// TwinCAT 3 PLC project SPS_Demonstrator
// ProgramVersion: 3.1.4026.21
// libraries:
//   Tc2_Standard, * (Beckhoff Automation GmbH)
//   Tc2_System, * (Beckhoff Automation GmbH)
//   Tc3_EventLogger, * (Beckhoff Automation GmbH)
//   Tc3_Module, * (Beckhoff Automation GmbH)
// project tree:
//   GVLs/ GVL.TcGVL, GVL_HRL.TcGVL, GVL_HRL_Sim.TcGVL, GVL_MBS.TcGVL, GVL_Sim.TcGVL, GVL_SST.TcGVL, GVL_VSG.TcGVL, GVL_VSG_Sim.TcGVL, OPCUA.TcGVL
//   / PlcTask.TcTTO
//   POUs/AtomicSkillsSchablonen/ AutomaticColorDetection_nichtfertig.TcPOU, AxisControl_Encoder.TcPOU, AxisControl_MultipleInputSensors.TcPOU, CompressorControl.TcPOU, CuttingProcess.TcPOU, HardeningProcess.TcPOU, SecuringWorkpiece.TcPOU, StampingProcess.TcPOU
//   POUs/ControlOfOutputs/ HRL_ControlOfOutputs.TcPOU, MBS_ControlOfOutputs.TcPOU, SST_ControlOfOutputs.TcPOU, VSG_ControlOfOutputs.TcPOU
//   POUs/DiagnosisHandler/ HRL_DiagnosisHandler.TcPOU, VSG_DiagnosisHandler.TcPOU
//   POUs/ HRL_SkillSet.TcPOU, MBS_SkillSet.TcPOU, SST_SkillSet.TcPOU, VSG_SkillSet.TcPOU
//   POUs/InitStateDrive/ HRL_RGB_InitialStateDrive.TcPOU, MBS_DmPD_InitialStateDrive.TcPOU, MBS_MR01_InitialStateDrive.TcPOU, MBS_MR02_InitialStateDrive.TcPOU, MBS_VSG_InitialStateDrive.TcPOU, SST_PD_InitialStateDrive.TcPOU, VSG_InitialStateDrive.TcPOU
//   POUs/MethodenBeispiele/ FB_MyOpcUaMethod.TcPOU, JobMethode_Schablone.TcPOU
//   POUs/Moduls/HRL_Skills/ HRL_CB_AS_HorizontalMoveSensors.TcPOU, HRL_NMethod_Auslagern.TcPOU, HRL_RGB_AS_HorizontalMoveEncoders.TcPOU, HRL_RGB_AS_HorizontalMoveSensors.TcPOU, HRL_RGB_AS_VerticalMoveEncoders.TcPOU
//   POUs/Moduls/MBS_Skills/ MBS_CB_AS_HorizontalMove.TcPOU, MBS_DmPD_AS_HorizontalMove.TcPOU, MBS_DmPD_AS_RotationMove.TcPOU, MBS_MR01_AS_HardeningProcess.TcPOU, MBS_MR01_AS_HorizontalMoveSensors.TcPOU, MBS_MR01_AS_SecuringProcess.TcPOU, MBS_MR02_AS_CuttingProcess.TcPOU, MBS_VSG_AS_HorizontalMove.TcPOU, MBS_VSG_AS_SuctionProcess.TcPOU, MBS_VSG_AS_VerticalMove.TcPOU
//   POUs/Moduls/SST_Skills/ SST_CB_AS_HorizontalMove.TcPOU, SST_CS_AS_ColorDetection.TcPOU, SST_PD_AS_HorizontalMove.TcPOU
//   POUs/Moduls/VSG_Skills/ VSG_AS_CompressorControl.TcPOU, VSG_AS_HorizontalMoveEncoder.TcPOU, VSG_AS_RotationMoveEncoder.TcPOU, VSG_AS_VerticalMoveEncoder.TcPOU
//   POUs/OperatingModes/ HRL_OperatingModes.TcPOU, VSG_OperatingModes.TcPOU, MBS_OperatingModes.TcPOU, SST_OperatingModes.TcPOU, VSG_OperatingModes_alt.TcPOU
// real-time tasks:
//   TASK PlcTask: cycle T#10ms, priority 20, ADS port 350
// I/O:
//   DEVICE Gerät 1 (EtherCAT), AmsNetId 5.152.132.139.2.1
//     Klemme 1 (EK1200) [EK1200-5000 EtherCAT Netzteil (2A E-Bus)]
//       Klemme 2 (EL1512) [EL1512 2K. +/- Zaehler 24V, 1kHz]
//       Klemme 3 (EL1512) [EL1512 2K. +/- Zaehler 24V, 1kHz]
//       Klemme 4 (EL1512) [EL1512 2K. +/- Zaehler 24V, 1kHz]
//       Klemme 5 (EL1512) [EL1512 2K. +/- Zaehler 24V, 1kHz]
//       Klemme 6 (EL1512) [EL1512 2K. +/- Zaehler 24V, 1kHz]
//       Klemme 7 (EL1409) [EL1409 16K. Dig. Eingang 24V, 3ms]
//       Klemme 8 (EL1409) [EL1409 16K. Dig. Eingang 24V, 3ms]
//       Klemme 9 (EL2409) [EL2409 16K. Dig. Ausgang 24V, 0.5A]
//       Klemme 10 (EL2409) [EL2409 16K. Dig. Ausgang 24V, 0.5A]
//       Klemme 11 (EL2008) [EL2008 8K. Dig. Ausgang 24V, 0.5A]
//       Klemme 12 (EL3072) [EL3072 2K. Ana. Eingang  +/-10V, +/-20mA]
//       Klemme 13 (EL9011) [EL9011 Endklemme]
// variable links:
//   SPS_Demonstrator/SPS_Demonstrator Instance <-> Device 1 (EtherCAT)/Term 1 (EK1200)/Term 10 (EL2409)
//     PlcTask Outputs/GVL_MBS.MBS_Kompressor <-> Channel 2/Output
//     PlcTask Outputs/GVL_MBS.MBS_Leuchte_Ofen <-> Channel 1/Output
//     PlcTask Outputs/GVL_MBS.MBS_MV_Ofentuer <-> Channel 5/Output
//     PlcTask Outputs/GVL_MBS.MBS_MV_Schieber <-> Channel 6/Output
//     PlcTask Outputs/GVL_MBS.MBS_MV_Vakuum <-> Channel 3/Output
//     PlcTask Outputs/GVL_MBS.MBS_MV_senken <-> Channel 4/Output
//     PlcTask Outputs/GVL_SST.SST_Kompressor <-> Channel 16/Output
//     PlcTask Outputs/GVL_SST.SST_MOT_Foerderband <-> Channel 15/Output
//     PlcTask Outputs/GVL_VSG.VSG_Kompressor <-> Channel 13/Output
//     PlcTask Outputs/GVL_VSG.VSG_MOT_drehen_CCW <-> Channel 12/Output
//     PlcTask Outputs/GVL_VSG.VSG_MOT_drehen_CW <-> Channel 11/Output
//     PlcTask Outputs/GVL_VSG.VSG_MOT_horizontal_rueckwaerts <-> Channel 9/Output
//     PlcTask Outputs/GVL_VSG.VSG_MOT_horizontal_vorwaerts <-> Channel 10/Output
//     PlcTask Outputs/GVL_VSG.VSG_MOT_vertikal_hoch <-> Channel 7/Output
//     PlcTask Outputs/GVL_VSG.VSG_MOT_vertikal_runter <-> Channel 8/Output
//     PlcTask Outputs/GVL_VSG.VSG_MV_Vakuum <-> Channel 14/Output
//   SPS_Demonstrator/SPS_Demonstrator Instance <-> Device 1 (EtherCAT)/Term 1 (EK1200)/Term 11 (EL2008)
//     PlcTask Outputs/GVL_SST.SST_MV_blau <-> Channel 3/Output
//     PlcTask Outputs/GVL_SST.SST_MV_rot <-> Channel 2/Output
//     PlcTask Outputs/GVL_SST.SST_MV_weiss <-> Channel 1/Output
//   SPS_Demonstrator/SPS_Demonstrator Instance <-> Device 1 (EtherCAT)/Term 1 (EK1200)/Term 12 (EL3072)
//     PlcTask Inputs/GVL_SST.SST_Farbsensor <-> AI Standard Channel 1/Value
//   SPS_Demonstrator/SPS_Demonstrator Instance <-> Device 1 (EtherCAT)/Term 1 (EK1200)/Term 2 (EL1512)
//     PlcTask Inputs/GVL_HRL.HRL_Enc_horizontal_I1 <-> CNT Inputs Channel 1/Counter value
//     PlcTask Inputs/GVL_HRL.HRL_Enc_horizontal_I2 <-> CNT Inputs Channel 2/Counter value
//     PlcTask Outputs/GVL_HRL.HRL_K1_1_Zaehler_Zuruecksetzen <-> CNT Outputs Channel 1/Control/Set counter
//   SPS_Demonstrator/SPS_Demonstrator Instance <-> Device 1 (EtherCAT)/Term 1 (EK1200)/Term 3 (EL1512)
//     PlcTask Inputs/GVL_HRL.HRL_Enc_vertikal_I1 <-> CNT Inputs Channel 1/Counter value
//     PlcTask Inputs/GVL_HRL.HRL_Enc_vertikal_I2 <-> CNT Inputs Channel 2/Counter value
//     PlcTask Outputs/GVL_HRL.HRL_K1_2_Zaehler_Zuruecksetzen <-> CNT Outputs Channel 1/Control/Set counter
//   SPS_Demonstrator/SPS_Demonstrator Instance <-> Device 1 (EtherCAT)/Term 1 (EK1200)/Term 4 (EL1512)
//     PlcTask Inputs/GVL_VSG.VSG_Enc_vertikal_I1 <-> CNT Inputs Channel 1/Counter value
//     PlcTask Inputs/GVL_VSG.VSG_Enc_vertikal_I2 <-> CNT Inputs Channel 2/Counter value
//     PlcTask Outputs/GVL_VSG.VSG_K1_3_Zaehler_Zuruecksetzen <-> CNT Outputs Channel 1/Control/Set counter
//   SPS_Demonstrator/SPS_Demonstrator Instance <-> Device 1 (EtherCAT)/Term 1 (EK1200)/Term 5 (EL1512)
//     PlcTask Inputs/GVL_VSG.VSG_Enc_horizontal_I1 <-> CNT Inputs Channel 1/Counter value
//     PlcTask Inputs/GVL_VSG.VSG_Enc_horizontal_I2 <-> CNT Inputs Channel 2/Counter value
//     PlcTask Outputs/GVL_VSG.VSG_K1_4_Zaehler_Zuruecksetzen <-> CNT Outputs Channel 1/Set counter
//   SPS_Demonstrator/SPS_Demonstrator Instance <-> Device 1 (EtherCAT)/Term 1 (EK1200)/Term 6 (EL1512)
//     PlcTask Inputs/GVL_VSG.VSG_Enc_drehen_I1 <-> CNT Inputs Channel 1/Counter value
//     PlcTask Inputs/GVL_VSG.VSG_Enc_drehen_I2 <-> CNT Inputs Channel 2/Counter value
//     PlcTask Outputs/GVL_VSG.VSG_K1_5_Zaehler_Zuruecksetzen <-> CNT Outputs Channel 1/Control/Set counter
//   SPS_Demonstrator/SPS_Demonstrator Instance <-> Device 1 (EtherCAT)/Term 1 (EK1200)/Term 7 (EL1409)
//     PlcTask Inputs/GVL_HRL.HRL_LS_aussen <-> DIP Inputs/Input Channel 3
//     PlcTask Inputs/GVL_HRL.HRL_LS_innen <-> DIP Inputs/Input Channel 2
//     PlcTask Inputs/GVL_HRL.HRL_Ref_Taster_Ausleger_hinten <-> DIP Inputs/Input Channel 8
//     PlcTask Inputs/GVL_HRL.HRL_Ref_Taster_Ausleger_vorne <-> DIP Inputs/Input Channel 7
//     PlcTask Inputs/GVL_HRL.HRL_Ref_Taster_horizontal <-> DIP Inputs/Input Channel 1
//     PlcTask Inputs/GVL_HRL.HRL_Ref_Taster_vertikal <-> DIP Inputs/Input Channel 4
//     PlcTask Inputs/GVL_HRL.HRL_Spursensor_1_unten <-> DIP Inputs/Input Channel 5
//     PlcTask Inputs/GVL_HRL.HRL_Spursensor_2_oben <-> DIP Inputs/Input Channel 6
//     PlcTask Inputs/GVL_MBS.MBS_LS_Ende_Foerderband <-> DIP Inputs/Input Channel 11
//     PlcTask Inputs/GVL_MBS.MBS_Ref_Taster_DK_Pos_Foerderband <-> DIP Inputs/Input Channel 10
//     PlcTask Inputs/GVL_MBS.MBS_Ref_Taster_DK_Pos_Saege <-> DIP Inputs/Input Channel 12
//     PlcTask Inputs/GVL_MBS.MBS_Ref_Taster_DK_Pos_Sauger <-> DIP Inputs/Input Channel 9
//     PlcTask Inputs/GVL_MBS.MBS_Ref_Taster_Ofenschieber_aussen <-> DIP Inputs/Input Channel 15
//     PlcTask Inputs/GVL_MBS.MBS_Ref_Taster_Ofenschieber_innen <-> DIP Inputs/Input Channel 14
//     PlcTask Inputs/GVL_MBS.MBS_Ref_Taster_Sauger_Pos_DK <-> DIP Inputs/Input Channel 13
//     PlcTask Inputs/GVL_MBS.MBS_Ref_Taster_Sauger_Pos_Ofen <-> DIP Inputs/Input Channel 16
//   SPS_Demonstrator/SPS_Demonstrator Instance <-> Device 1 (EtherCAT)/Term 1 (EK1200)/Term 8 (EL1409)
//     PlcTask Inputs/GVL.diNotAus_Kanal_A <-> DIP Inputs/Input Channel 11
//     PlcTask Inputs/GVL.diNotAus_Kanal_B <-> DIP Inputs/Input Channel 12
//     PlcTask Inputs/GVL_MBS.MBS_LS_Ofen <-> DIP Inputs/Input Channel 1
//     PlcTask Inputs/GVL_SST.SST_Impulstaster <-> DIP Inputs/Input Channel 5
//     PlcTask Inputs/GVL_SST.SST_LS_Eingang <-> DIP Inputs/Input Channel 6
//     PlcTask Inputs/GVL_SST.SST_LS_blau <-> DIP Inputs/Input Channel 10
//     PlcTask Inputs/GVL_SST.SST_LS_nach_Farbsensor <-> DIP Inputs/Input Channel 7
//     PlcTask Inputs/GVL_SST.SST_LS_rot <-> DIP Inputs/Input Channel 9
//     PlcTask Inputs/GVL_SST.SST_LS_weiss <-> DIP Inputs/Input Channel 8
//     PlcTask Inputs/GVL_VSG.VSG_Ref_Schalter_drehen <-> DIP Inputs/Input Channel 4
//     PlcTask Inputs/GVL_VSG.VSG_Ref_Schalter_horizontal <-> DIP Inputs/Input Channel 3
//     PlcTask Inputs/GVL_VSG.VSG_Ref_Schalter_vertikal <-> DIP Inputs/Input Channel 2
//   SPS_Demonstrator/SPS_Demonstrator Instance <-> Device 1 (EtherCAT)/Term 1 (EK1200)/Term 9 (EL2409)
//     PlcTask Outputs/GVL_HRL.HRL_MOT_Ausleger_rueckwaerts <-> Channel 8/Output
//     PlcTask Outputs/GVL_HRL.HRL_MOT_Ausleger_vorwaerts <-> Channel 7/Output
//     PlcTask Outputs/GVL_HRL.HRL_MOT_Foerderband_rueckwaerts <-> Channel 2/Output
//     PlcTask Outputs/GVL_HRL.HRL_MOT_Foerderband_vorwaerts <-> Channel 1/Output
//     PlcTask Outputs/GVL_HRL.HRL_MOT_horizontal_zum_Foerderband <-> Channel 4/Output
//     PlcTask Outputs/GVL_HRL.HRL_MOT_horizontal_zum_Regal <-> Channel 3/Output
//     PlcTask Outputs/GVL_HRL.HRL_MOT_vertikal_hoch <-> Channel 6/Output
//     PlcTask Outputs/GVL_HRL.HRL_MOT_vertikal_runter <-> Channel 5/Output
//     PlcTask Outputs/GVL_MBS.MBS_MOT_DK_CCW <-> Channel 10/Output
//     PlcTask Outputs/GVL_MBS.MBS_MOT_DK_CW <-> Channel 9/Output
//     PlcTask Outputs/GVL_MBS.MBS_MOT_Foerderband_vorwaerts <-> Channel 11/Output
//     PlcTask Outputs/GVL_MBS.MBS_MOT_Ofenschieber_ausfahren <-> Channel 14/Output
//     PlcTask Outputs/GVL_MBS.MBS_MOT_Ofenschieber_einfahren <-> Channel 13/Output
//     PlcTask Outputs/GVL_MBS.MBS_MOT_Saege <-> Channel 12/Output
//     PlcTask Outputs/GVL_MBS.MBS_MOT_Sauger_zum_DK <-> Channel 16/Output
//     PlcTask Outputs/GVL_MBS.MBS_MOT_Sauger_zum_Ofen <-> Channel 15/Output

CONFIGURATION SPS_Demonstrator
    RESOURCE PLC ON TwinCAT3
        TASK PlcTask(INTERVAL := T#10ms, PRIORITY := 20);
        PROGRAM HRL_SkillSet WITH PlcTask : HRL_SkillSet;
        PROGRAM VSG_SkillSet WITH PlcTask : VSG_SkillSet;
    END_RESOURCE
END_CONFIGURATION

// ---- GVLs/GVL.TcGVL
{attribute 'qualified_only'}
VAR_GLOBAL
	// xDI%139.2_S1_2
	diNotAus_Kanal_A AT %I*: BOOL;
	// xDI%139.3_S1_2
	diNotAus_Kanal_B AT %I*: BOOL;
END_VAR

// ---- GVLs/GVL_HRL.TcGVL
{attribute 'qualified_only'}
VAR_GLOBAL
	// udiDI%41.0_A2_5
	{attribute 'OPC.UA.DA' := '1'} // für OPC UA freigeben
	HRL_Enc_horizontal_I1 AT %I*: UDINT;
	{attribute 'OPC.UA.DA' := '1'} // für OPC UA freigeben
	// udiDI%47.0_A2_5
	HRL_Enc_horizontal_I2 AT %I*: UDINT;
	{attribute 'OPC.UA.DA' := '1'} // für OPC UA freigeben
	// udiDI%53.0_A2_5
	HRL_Enc_vertikal_I1 AT %I*: UDINT;
	{attribute 'OPC.UA.DA' := '1'} // für OPC UA freigeben
	// udiDI%59.0_A2_5
	HRL_Enc_vertikal_I2 AT %I*: UDINT;
	{attribute 'OPC.UA.DA' := '1'} // für OPC UA freigeben
	// xDI%136.0_A2_2
	HRL_Ref_Taster_horizontal AT %I*: BOOL;
	{attribute 'OPC.UA.DA' := '1'} // für OPC UA freigeben
	// xDI%136.1_A2_1
	{attribute 'OPC.UA.DA' := '1'} // für OPC UA freigeben
	HRL_LS_innen AT %I*: BOOL;
	// xDI%136.2_A2_1
	{attribute 'OPC.UA.DA' := '1'} // für OPC UA freigeben
	HRL_LS_aussen AT %I*: BOOL;
	// xDI%136.3_A2_2
	{attribute 'OPC.UA.DA' := '1'} // für OPC UA freigeben
	HRL_Ref_Taster_vertikal AT %I*: BOOL;
	// xDI%136.4_A2_3
	{attribute 'OPC.UA.DA' := '1'} // für OPC UA freigeben
	HRL_Spursensor_1_unten AT %I*: BOOL;
	// xDI%136.5_A2_3
	{attribute 'OPC.UA.DA' := '1'} // für OPC UA freigeben
	HRL_Spursensor_2_oben AT %I*: BOOL;
	// xDI%136.6_A2_2
	{attribute 'OPC.UA.DA' := '1'} // für OPC UA freigeben
	HRL_Ref_Taster_Ausleger_vorne AT %I*: BOOL;
	// xDI%136.7_A2_2
	{attribute 'OPC.UA.DA' := '1'} // für OPC UA freigeben
	HRL_Ref_Taster_Ausleger_hinten AT %I*: BOOL;
	// xDO%111.0_A2_2	
	{attribute 'OPC.UA.DA' := '1'} // für OPC UA freigeben
	HRL_MOT_Foerderband_vorwaerts AT %Q*: BOOL;
	// xDO%111.1_A2_2
	{attribute 'OPC.UA.DA' := '1'} // für OPC UA freigeben
	HRL_MOT_Foerderband_rueckwaerts AT %Q*: BOOL;
	// xDO%111.2_A2_4
	{attribute 'OPC.UA.DA' := '1'} // für OPC UA freigeben
	HRL_MOT_horizontal_zum_Regal AT %Q*: BOOL;
	// xDO%111.3_A2_4
	{attribute 'OPC.UA.DA' := '1'} // für OPC UA freigeben
	HRL_MOT_horizontal_zum_Foerderband AT %Q*: BOOL;
	// xDO%111.4_A2_4
	{attribute 'OPC.UA.DA' := '1'} // für OPC UA freigeben
	HRL_MOT_vertikal_runter AT %Q*: BOOL;
	// xDO%111.5_A2_4
	{attribute 'OPC.UA.DA' := '1'} // für OPC UA freigeben
	HRL_MOT_vertikal_hoch AT %Q*: BOOL;
	// xDO%111.6_A2_4
	{attribute 'OPC.UA.DA' := '1'} // für OPC UA freigeben
	HRL_MOT_Ausleger_vorwaerts AT %Q*: BOOL;
	// xDO%111.7_A2_4
	{attribute 'OPC.UA.DA' := '1'} // für OPC UA freigeben
	HRL_MOT_Ausleger_rueckwaerts AT %Q*: BOOL;
	{attribute 'OPC.UA.DA' := '1'} // für OPC UA freigeben
	HRL_K1_1_Zaehler_Zuruecksetzen AT %Q*: BOOL;
	{attribute 'OPC.UA.DA' := '1'} // für OPC UA freigeben
	HRL_K1_2_Zaehler_Zuruecksetzen AT %Q*: BOOL;
END_VAR

// ---- GVLs/GVL_HRL_Sim.TcGVL
{attribute 'qualified_only'}
VAR_GLOBAL
	// Spiegel von GVL_HRL (Eingänge)
    HRL_Enc_horizontal_I1 : UDINT;
	// udiDI%47.0_A2_5
	HRL_Enc_horizontal_I2 : UDINT;
	// udiDI%53.0_A2_5
	HRL_Enc_vertikal_I1 : UDINT;
	// udiDI%59.0_A2_5
	HRL_Enc_vertikal_I2 : UDINT;
	// xDI%136.0_A2_2
	HRL_Ref_Taster_horizontal : BOOL;
	// xDI%136.1_A2_1
	HRL_LS_innen : BOOL;
	// xDI%136.2_A2_1
	HRL_LS_aussen : BOOL;
	// xDI%136.3_A2_2
	HRL_Ref_Taster_vertikal : BOOL;
	// xDI%136.4_A2_3
	HRL_Spursensor_1_unten : BOOL;
	// xDI%136.5_A2_3
	HRL_Spursensor_2_oben : BOOL;
	// xDI%136.6_A2_2
	HRL_Ref_Taster_Ausleger_vorne : BOOL;
	// xDI%136.7_A2_2
	HRL_Ref_Taster_Ausleger_hinten : BOOL;
	// xDO%111.0_A2_2	
	HRL_MOT_Foerderband_vorwaerts : BOOL;
	// xDO%111.1_A2_2
	HRL_MOT_Foerderband_rueckwaerts : BOOL;
	// xDO%111.2_A2_4
	HRL_MOT_horizontal_zum_Regal : BOOL;
	// xDO%111.3_A2_4
	HRL_MOT_horizontal_zum_Foerderband : BOOL;
	// xDO%111.4_A2_4
	HRL_MOT_vertikal_runter : BOOL;
	// xDO%111.5_A2_4
	HRL_MOT_vertikal_hoch : BOOL;
	// xDO%111.6_A2_4
	HRL_MOT_Ausleger_vorwaerts : BOOL;
	// xDO%111.7_A2_4
	HRL_MOT_Ausleger_rueckwaerts : BOOL;
	HRL_K1_1_Zaehler_Zuruecksetzen : BOOL;
	HRL_K1_2_Zaehler_Zuruecksetzen : BOOL;
END_VAR

// ---- GVLs/GVL_MBS.TcGVL
{attribute 'qualified_only'}
VAR_GLOBAL
	// xDI%137.0_A3_2
	MBS_Ref_Taster_DK_Pos_Sauger AT %I*: BOOL;
	// xDI%137.1_A3_2
	MBS_Ref_Taster_DK_Pos_Foerderband AT %I*: BOOL;
	// xDI%137.2_A3_1
	MBS_LS_Ende_Foerderband AT %I*: BOOL;
	// xDI%137.3_A3_2
	MBS_Ref_Taster_DK_Pos_Saege AT %I*: BOOL;
	// xDI%137.4_A3_2
	MBS_Ref_Taster_Sauger_Pos_DK AT %I*: BOOL;
	// xDI%137.5_A3_2
	MBS_Ref_Taster_Ofenschieber_innen AT %I*: BOOL;
	// xDI%137.6_A3_2
	MBS_Ref_Taster_Ofenschieber_aussen AT %I*: BOOL;
	// xDI%137.7_A3_2
	MBS_Ref_Taster_Sauger_Pos_Ofen AT %I*: BOOL;
	// xDI%138.0_A3_1
	MBS_LS_Ofen AT %I*: BOOL;
	// xDO%112.0_A3_4
	MBS_MOT_DK_CW AT %Q*: BOOL;
	// xDO%112.1_A3_4
	MBS_MOT_DK_CCW AT %Q*: BOOL;
	// xDO%112.2_A3_2
	MBS_MOT_Foerderband_vorwaerts AT %Q*: BOOL;
	// xDO%112.3_A3_6
	MBS_MOT_Saege AT %Q*: BOOL;
	// xDO%112.4_A3_3
	MBS_MOT_Ofenschieber_einfahren AT %Q*: BOOL;
	// xDO%112.5_A3_3
	MBS_MOT_Ofenschieber_ausfahren AT %Q*: BOOL;
	// xDO%112.6_A3_5
	MBS_MOT_Sauger_zum_Ofen AT %Q*: BOOL;
	// xDO%112.7_A3_5
	MBS_MOT_Sauger_zum_DK AT %Q*: BOOL;
	// xDO%113.0_A3_7
	MBS_Leuchte_Ofen AT %Q*: BOOL;
	// xDO%113.1_A3_8
	MBS_Kompressor AT %Q*: BOOL;
	// xDO%113.2_A3_5
	MBS_MV_Vakuum AT %Q*: BOOL;
	// xDO%113.3_A3_5
	MBS_MV_senken AT %Q*: BOOL;
	// xDO%113.4_A3_5
	MBS_MV_Ofentuer AT %Q*: BOOL;
	// xDO%113.5_A3_5
	MBS_MV_Schieber AT %Q*: BOOL;
END_VAR

// ---- GVLs/GVL_Sim.TcGVL
{attribute 'qualified_only'}
VAR_GLOBAL
	bSimMode : BOOL ;   // FALSE = reale Hardware, TRUE = Python-Simulation

    // Spiegel von GVL
    diNotAus_Kanal_A : BOOL ;
    diNotAus_Kanal_B : BOOL ;
    
END_VAR

// ---- GVLs/GVL_SST.TcGVL
{attribute 'qualified_only'}
VAR_GLOBAL
	// xDO%115.0_A5_5
	SST_MV_weiss AT %Q*: BOOL;
	// xDO%115.1_A5_5
	SST_MV_rot AT %Q*: BOOL;
	// xDO%115.2_A5_5
	SST_MV_blau AT %Q*: BOOL;
	// iAI%130.0_A5_4
	SST_Farbsensor AT %I*: INT;
	// xDI%138.4_A5_1
	SST_Impulstaster AT %I*: BOOL;
	// xDI%138.5_A5_1
	SST_LS_Eingang AT %I*: BOOL;
	// xDI%138.6_A5_1
	SST_LS_nach_Farbsensor AT %I*: BOOL;
	// xDI%138.7_A5_1
	SST_LS_weiss AT %I*: BOOL;
	// xDI%139.0_A5_1
	SST_LS_rot AT %I*: BOOL;
	// xDI%139.1_A5_1
	SST_LS_blau AT %I*: BOOL;
	// xDO%114.6_A5_2
	SST_MOT_Foerderband AT %Q*: BOOL;
	// xDO%114.7_A5_8
	SST_Kompressor AT %Q*: BOOL;
END_VAR

// ---- GVLs/GVL_VSG.TcGVL
{attribute 'qualified_only'}
VAR_GLOBAL
	// udiDI%65.0_A4_5
	{attribute 'OPC.UA.DA' := '1'} // für OPC UA freigeben
	VSG_Enc_vertikal_I1 AT %I*: UDINT;
	{attribute 'OPC.UA.DA' := '1'} // für OPC UA freigeben
	// udiDI%71.0_A4_5
	VSG_Enc_vertikal_I2 AT %I*: UDINT;
	{attribute 'OPC.UA.DA' := '1'} // für OPC UA freigeben
	// udiDI%77.0_A4_5
	VSG_Enc_horizontal_I1 AT %I*: UDINT;
	{attribute 'OPC.UA.DA' := '1'} // für OPC UA freigeben
	// udiDI%83.0_A4_5
	VSG_Enc_horizontal_I2 AT %I*: UDINT;
	{attribute 'OPC.UA.DA' := '1'} // für OPC UA freigeben
	// udiDI%89.0_A4_5
	VSG_Enc_drehen_I1 AT %I*: UDINT;
	{attribute 'OPC.UA.DA' := '1'} // für OPC UA freigeben
	// udiDI%95.0_A4_5
	VSG_Enc_drehen_I2 AT %I*: UDINT;
	{attribute 'OPC.UA.DA' := '1'} // für OPC UA freigeben
	// xDI%138.1_A4_2
	VSG_Ref_Schalter_vertikal AT %I*: BOOL;
	{attribute 'OPC.UA.DA' := '1'} // für OPC UA freigeben
	// xDI%138.2_A4_2
	VSG_Ref_Schalter_horizontal AT %I*: BOOL;
	{attribute 'OPC.UA.DA' := '1'} // für OPC UA freigeben
	// xDI%138.3_A4_2
	VSG_Ref_Schalter_drehen AT %I*: BOOL;
	{attribute 'OPC.UA.DA' := '1'} // für OPC UA freigeben
	// xDO%113.6_A4_4
	VSG_MOT_vertikal_hoch AT %Q*: BOOL;
	{attribute 'OPC.UA.DA' := '1'} // für OPC UA freigeben
	// xDO%113.7_A4_4
	VSG_MOT_vertikal_runter AT %Q*: BOOL;
	{attribute 'OPC.UA.DA' := '1'} // für OPC UA freigeben
	// xDO%114.0_A4_4
	VSG_MOT_horizontal_rueckwaerts AT %Q*: BOOL;
	{attribute 'OPC.UA.DA' := '1'} // für OPC UA freigeben
	// xDO%114.1_A4_4
	VSG_MOT_horizontal_vorwaerts AT %Q*: BOOL;
	{attribute 'OPC.UA.DA' := '1'} // für OPC UA freigeben
	// xDO%114.2_A4_4
	VSG_MOT_drehen_CW AT %Q*: BOOL;
	{attribute 'OPC.UA.DA' := '1'} // für OPC UA freigeben
	// xDO%114.3_A4_4
	VSG_MOT_drehen_CCW AT %Q*: BOOL;
	{attribute 'OPC.UA.DA' := '1'} // für OPC UA freigeben
	// xDO%114.4_A4_8
	VSG_Kompressor AT %Q*: BOOL;
	{attribute 'OPC.UA.DA' := '1'} // für OPC UA freigeben
	// xDO%114.5_A4_5
	{attribute 'OPC.UA.DA' := '1'} // für OPC UA freigeben
	VSG_MV_Vakuum AT %Q*: BOOL;
	{attribute 'OPC.UA.DA' := '1'} // für OPC UA freigeben
	VSG_K1_4_Zaehler_Zuruecksetzen AT %Q*: BOOL;
	{attribute 'OPC.UA.DA' := '1'} // für OPC UA freigeben
	VSG_K1_5_Zaehler_Zuruecksetzen AT %Q*: BOOL;
	{attribute 'OPC.UA.DA' := '1'} // für OPC UA freigeben
	VSG_K1_3_Zaehler_Zuruecksetzen AT %Q*: BOOL;
END_VAR

// ---- GVLs/GVL_VSG_Sim.TcGVL
{attribute 'qualified_only'}
VAR_GLOBAL
    // Simulierte VSG Eingänge
    VSG_Enc_vertikal_I1 : UDINT;
    VSG_Enc_vertikal_I2 : UDINT;

    VSG_Enc_horizontal_I1 : UDINT;
    VSG_Enc_horizontal_I2 : UDINT;

    VSG_Enc_drehen_I1 : UDINT;
    VSG_Enc_drehen_I2 : UDINT;

    VSG_Ref_Schalter_vertikal : BOOL;
    VSG_Ref_Schalter_horizontal : BOOL;
    VSG_Ref_Schalter_drehen : BOOL;

    // Simulierte VSG Ausgänge
    VSG_MOT_vertikal_hoch : BOOL;
    VSG_MOT_vertikal_runter : BOOL;

    VSG_MOT_horizontal_vorwaerts : BOOL;
    VSG_MOT_horizontal_rueckwaerts : BOOL;

    VSG_MOT_drehen_CW : BOOL;
    VSG_MOT_drehen_CCW : BOOL;

    VSG_Kompressor : BOOL;
    VSG_MV_Vakuum : BOOL;

    VSG_K1_4_Zaehler_Zuruecksetzen : BOOL;
    VSG_K1_5_Zaehler_Zuruecksetzen : BOOL;
    VSG_K1_3_Zaehler_Zuruecksetzen : BOOL;
END_VAR

// ---- GVLs/OPCUA.TcGVL
{attribute 'qualified_only'}
VAR_GLOBAL
	{attribute 'OPC.UA.DA' := '1'} // für OPC UA freigeben
	TriggerD1 : BOOL := FALSE;
	{attribute 'OPC.UA.DA' := '1'} // für OPC UA freigeben
	TriggerD2 : BOOL := FALSE;
	{attribute 'OPC.UA.DA' := '1'} // für OPC UA freigeben
	TriggerD3 : BOOL := FALSE;
	{attribute 'OPC.UA.DA' := '1'} // für OPC UA freigeben
    {attribute 'OPC.UA.DA.Access' := '3'} // Read/Write
	Alt_found : BOOL := FALSE;
	{attribute 'OPC.UA.DA' := '1'} // für OPC UA freigeben
    {attribute 'OPC.UA.DA.Access' := '3'} // Read/Write
	Alt_abort : BOOL := FALSE;
	{attribute 'OPC.UA.DA' := '1'} // für OPC UA freigeben
    {attribute 'OPC.UA.DA.Access' := '3'} // Read/Write
	Diag_finished : BOOL := FALSE;
	{attribute 'OPC.UA.DA' := '1'} // für OPC UA freigeben
    {attribute 'OPC.UA.DA.Access' := '3'} // Read/Write
	Cycle_finished : BOOL := FALSE;
	{attribute 'OPC.UA.DA' := '1'}
    LastGEMMAStateBeforeFailure: STRING;
	{attribute 'OPC.UA.DA' := '1'}
    lastExecutedSkill: STRING := '';
	{attribute 'OPC.UA.DA' := '1'}
	{attribute 'OPC.UA.DA.Access' := '3'} // Read/Write
    lastFinishedSkill: STRING := '';
	{attribute 'OPC.UA.DA' := '1'}
    lastExecutedProcess: STRING := '';
END_VAR

// ---- POUs/HRL_SkillSet.TcPOU
PROGRAM HRL_SkillSet
VAR
//Hochregallager Skillset	
	//HRL CombinedSkill_Auslagerung
	{attribute 'OPC.UA.DA':= '1'}
	HRL_NMethod_Auslagern : HRL_NMethod_Auslagern;
	bAuslagernAktiv : BOOL := FALSE;
	//HRL Conveyorbelt Skills
	{attribute 'OPC.UA.DA':= '1'}
	HRL_Skill_CB_MoveForwards: HRL_CB_AS_HorizontalMoveSensors; //Movement to Store-Out some goods on the Conveyorbelt
	{attribute 'OPC.UA.DA':= '1'}
	HRL_Skill_CB_MoveBackwards : HRL_CB_AS_HorizontalMoveSensors; //Movement to Store-In some goods on the Conveyorbelt
	
	//HRL RGB Skills
	{attribute 'OPC.UA.DA':= '1'}
	HRL_Skill_RGB_MoveBackwards : HRL_RGB_AS_HorizontalMoveSensors;	
	{attribute 'OPC.UA.DA':= '1'}
	HRL_Skill_RGB_MoveForwards : HRL_RGB_AS_HorizontalMoveSensors;	
	{attribute 'OPC.UA.DA':= '1'}
	HRL_Skill_RGB_MoveVerticalForwards : HRL_RGB_AS_VerticalMoveEncoders;	
	{attribute 'OPC.UA.DA':= '1'}
	HRL_Skill_RGB_MoveVerticalBackwards : HRL_RGB_AS_VerticalMoveEncoders;
	{attribute 'OPC.UA.DA':= '1'}
	HRL_Skill_RGB_MoveHorizontalForwards : HRL_RGB_AS_HorizontalMoveEncoders;	
	{attribute 'OPC.UA.DA':= '1'}
	HRL_Skill_RGB_MoveHorizontalBackwards : HRL_RGB_AS_HorizontalMoveEncoders;
	
	//Organisation FBs
	HRL_ControlOfOutputs : HRL_ControlOfOutputs;
	HRL_OperatingModes : HRL_OperatingModes;
	HRL_DiagnosisHandler : HRL_DiagnosisHandler;
	bAuslagernTrackingLatched : BOOL := FALSE;
	
	//InitialStateDrives
	HRL_RGB_InitialStateDrive : HRL_RGB_InitialStateDrive;
	
	
//Variablen zur Outputsteuerung
	HRL_CB_forwards : BOOL; //GVL_HRL.HRL_MOT_Foerderband_vorwaerts
	HRL_CB_backwards : BOOL; //GVL_HRL.HRL_MOT_Foerderband_rueckwaerts
	HRL_RGB_Forwards01 : BOOL; //GVL_HRL.HRL_MOT_Ausleger_vorwaerts
	HRL_RGB_Forwards02 : BOOL; //GVL_HRL.HRL_MOT_Ausleger_vorwaerts
	HRL_RGB_Backwards01 : BOOL; //GVL_HRL.HRL_MOT_Ausleger_rueckwaerts
	HRL_RGB_Backwards02 : BOOL; //GVL_HRL.HRL_MOT_Ausleger_rueckwaerts	
	HRL_RGB_VertikalDown01 : BOOL; //GVL_HRL.HRL_MOT_vertikal_runter		
	HRL_RGB_VertikalDown02 : BOOL; //GVL_HRL.HRL_MOT_vertikal_runter
	HRL_RGB_VertikalUp01 : BOOL; //GVL_HRL.HRL_MOT_vertikal_hoch
	HRL_RGB_VertikalUp02 : BOOL; //GVL_HRL.HRL_MOT_vertikal_hoch
	HRL_RGB_HorizontalForwards01 : BOOL; //GVL_HRL.HRL_MOT_horizontal_zum_Regal	
	HRL_RGB_HorizontalForwards02 : BOOL; //GVL_HRL.HRL_MOT_horizontal_zum_Regal	
	HRL_RGB_HorizontalBackwards01 : BOOL; //GVL_HRL.HRL_MOT_horizontal_zum_Foerderband
	HRL_RGB_HorizontalBackwards02 : BOOL; //GVL_HRL.HRL_MOT_horizontal_zum_Foerderband
//OutputVariablen für Init-Fahrt	
	Init_SRM_MotorBackwards : BOOL;
	Init_SRM_MotorForwards : BOOL;
	Init_RGB_VerticalUp : BOOL;
	Init_RGB_VerticalDown : BOOL;
	Init_RGB_HorizontalForwards : BOOL;
	Init_RGB_HorizontalBackwards : BOOL;
	
//Time Constraints
	TIME_TSR : TIME := T#150MS;
//Encoder Values for InitialStateDrive
	HRL_RGB_ET_Vertical01 : UDINT;
	HRL_RGB_ET_Vertical02 : UDINT;
	HRL_RGB_ET_Horizontall01 : UDINT;
	HRL_RGB_ET_Horizontall02 : UDINT;
	
	//GEMMA_Mappings
	sCurrentGemmaState : STRING(80) := '';
    sLastNonFailureGemmaState : STRING(80) := '';
    rtD2 : R_TRIG;
END_VAR

VAR_INPUT
	//Variablensetzung: Sollte später über SkillOA eingesetzt werden ODER Hard in SPS codiert (Diskussionspunkt)
	ResetButton: BOOL;
	StartButton: BOOL;
	ConfirmationButton: BOOL;
END_VAR

(* === Simulations-Override *)
IF GVL_Sim.bSimMode THEN
    GVL.diNotAus_Kanal_A                  := GVL_Sim.diNotAus_Kanal_A;
    GVL.diNotAus_Kanal_B                  := GVL_Sim.diNotAus_Kanal_B;
    GVL_HRL.HRL_Enc_horizontal_I1          := GVL_HRL_Sim.HRL_Enc_horizontal_I1;
    GVL_HRL.HRL_Enc_horizontal_I2          := GVL_HRL_Sim.HRL_Enc_horizontal_I2;
    GVL_HRL.HRL_Enc_vertikal_I1            := GVL_HRL_Sim.HRL_Enc_vertikal_I1;
    GVL_HRL.HRL_Enc_vertikal_I2            := GVL_HRL_Sim.HRL_Enc_vertikal_I2;
    // GVL_HRL - Digitaleingänge (BOOL)
    GVL_HRL.HRL_Ref_Taster_horizontal      := GVL_HRL_Sim.HRL_Ref_Taster_horizontal;
    GVL_HRL.HRL_LS_innen                   := GVL_HRL_Sim.HRL_LS_innen;
    GVL_HRL.HRL_LS_aussen                  := GVL_HRL_Sim.HRL_LS_aussen;
    GVL_HRL.HRL_Ref_Taster_vertikal        := GVL_HRL_Sim.HRL_Ref_Taster_vertikal;
    GVL_HRL.HRL_Spursensor_1_unten         := GVL_HRL_Sim.HRL_Spursensor_1_unten;
    GVL_HRL.HRL_Spursensor_2_oben          := GVL_HRL_Sim.HRL_Spursensor_2_oben;
    GVL_HRL.HRL_Ref_Taster_Ausleger_vorne  := GVL_HRL_Sim.HRL_Ref_Taster_Ausleger_vorne;
    GVL_HRL.HRL_Ref_Taster_Ausleger_hinten := GVL_HRL_Sim.HRL_Ref_Taster_Ausleger_hinten;
END_IF
(* ============================================================================= *)
HRL_OperatingModes(
    Start := StartButton,
    Stop := NOT (((GVL.diNotAus_Kanal_A) AND (GVL.diNotAus_Kanal_B))),
    Reset := ResetButton,
    Schalter := ConfirmationButton,
    Schrittkette_GS := ((HRL_RGB_InitialStateDrive.ResetMethodCall_SRM) AND (HRL_RGB_InitialStateDrive.ResetMethodCall_RGB_Horizontal) AND (HRL_RGB_InitialStateDrive.ResetMethodCall_RGB_Vertical)),
    Count1 := HRL_RGB_InitialStateDrive.Count_SRM_MotorBackw,
    Count2 := HRL_RGB_InitialStateDrive.Count_SRM_MotorForw,
    Alt_abort := OPCUA.Alt_abort,
    Err_detected := HRL_DiagnosisHandler.Err_detected,
    Diag_finished := HRL_DiagnosisHandler.Diag_finished,
    Alt_found := HRL_DiagnosisHandler.Alt_found,
    Cycle_finished := OPCUA.Cycle_finished
);


HRL_NMethod_Auslagern(
    ESS_OK := ((GVL.diNotAus_Kanal_A) AND (GVL.diNotAus_Kanal_B)),
    AutomaticMode := HRL_OperatingModes.F1,

    HRL_Enc_horizontal_I1 := GVL_HRL.HRL_Enc_horizontal_I1,
    HRL_Enc_horizontal_I2 := GVL_HRL.HRL_Enc_horizontal_I2,
    HRL_Enc_vertikal_I1 := GVL_HRL.HRL_Enc_vertikal_I1,
    HRL_Enc_vertikal_I2 := GVL_HRL.HRL_Enc_vertikal_I2,

    HRL_Ref_Taster_horizontal := GVL_HRL.HRL_Ref_Taster_horizontal,
    HRL_Ref_Taster_vertikal := GVL_HRL.HRL_Ref_Taster_vertikal,
    HRL_Ref_Taster_Ausleger_vorne := GVL_HRL.HRL_Ref_Taster_Ausleger_vorne,
    HRL_Ref_Taster_Ausleger_hinten := GVL_HRL.HRL_Ref_Taster_Ausleger_hinten,

    HRL_LS_innen := GVL_HRL.HRL_LS_innen,
    HRL_LS_aussen := GVL_HRL.HRL_LS_aussen
);

HRL_DiagnosisHandler(
    Diagnose_gefordert := HRL_OperatingModes.D2,
    ErrorDetectedRaw := HRL_NMethod_Auslagern.Error,
    Reset := ResetButton
);

HRL_RGB_InitialStateDrive(
    MethodCall_InitDrive := HRL_OperatingModes.MethodCall_InitStateDrive,
    ESS := ((GVL.diNotAus_Kanal_A) AND (GVL.diNotAus_Kanal_B)),
    InputInitDriveMode := HRL_OperatingModes.InputVar_InitStateDrive,
    TouchSensor01_SRM := GVL_HRL.HRL_Ref_Taster_Ausleger_hinten,
    TouchSensor02_RGB_vertical := GVL_HRL.HRL_Ref_Taster_vertikal,
    TouchSensor03_RGB_horizontal := GVL_HRL.HRL_Ref_Taster_horizontal,
    TOF_Time_TSR := TIME_TSR,
    InitDriveMode := HRL_OperatingModes.A6
);
Init_SRM_MotorBackwards := HRL_RGB_InitialStateDrive.SRM_MotorBackwards;
HRL_Skill_CB_MoveForwards(
    ESS := ((GVL.diNotAus_Kanal_A) AND (GVL.diNotAus_Kanal_B)),
    LightBarrierSensor_01 := GVL_HRL.HRL_LS_innen,
    LightBarrierSensor_02 := GVL_HRL.HRL_LS_aussen,
    AutomaticMode := HRL_OperatingModes.F1
);
HRL_CB_forwards := HRL_Skill_CB_MoveForwards.DO_MovingConveyorBelt;
HRL_Skill_CB_MoveBackwards(
    ESS := ((GVL.diNotAus_Kanal_A) AND (GVL.diNotAus_Kanal_B)),
    LightBarrierSensor_01 := GVL_HRL.HRL_LS_aussen,
    LightBarrierSensor_02 := GVL_HRL.HRL_LS_innen,
    AutomaticMode := HRL_OperatingModes.F1
);
HRL_CB_backwards := HRL_Skill_CB_MoveBackwards.DO_MovingConveyorBelt;
HRL_Skill_RGB_MoveForwards(
    ESS := ((GVL.diNotAus_Kanal_A) AND (GVL.diNotAus_Kanal_B)),
    TouchSensor01 := GVL_HRL.HRL_Ref_Taster_Ausleger_hinten,
    TouchSensor02 := GVL_HRL.HRL_Ref_Taster_Ausleger_vorne,
    TOF_Time_TSR := TIME_TSR,
    AutomaticMode := HRL_OperatingModes.F1
);
HRL_RGB_Forwards01 := HRL_Skill_RGB_MoveForwards.DO_MovingHorizontalRGB_01;
HRL_Skill_RGB_MoveBackwards(
    ESS := ((GVL.diNotAus_Kanal_A) AND (GVL.diNotAus_Kanal_B)),
    TouchSensor01 := GVL_HRL.HRL_Ref_Taster_Ausleger_vorne,
    TouchSensor02 := GVL_HRL.HRL_Ref_Taster_Ausleger_hinten,
    TOF_Time_TSR := TIME_TSR,
    AutomaticMode := HRL_OperatingModes.F1
);
HRL_RGB_Backwards01 := HRL_Skill_RGB_MoveBackwards.DO_MovingHorizontalRGB_01;
HRL_Skill_RGB_MoveVerticalForwards(
    ESS := ((GVL.diNotAus_Kanal_A) AND (GVL.diNotAus_Kanal_B)),
    TouchSensor01 := GVL_HRL.HRL_Ref_Taster_vertikal,
    EncoderStartPosition01 := GVL_HRL.HRL_Enc_vertikal_I1,
    EncoderStartPosition02 := GVL_HRL.HRL_Enc_vertikal_I2,
    TOF_TSR_TIME := TIME_TSR,
    AutomaticMode := HRL_OperatingModes.F1
);
HRL_RGB_VertikalDown01 := HRL_Skill_RGB_MoveVerticalForwards.DO_MovingVerticalRGB_01;
HRL_Skill_RGB_MoveVerticalBackwards(
    ESS := ((GVL.diNotAus_Kanal_A) AND (GVL.diNotAus_Kanal_B)),
    TouchSensor01 := GVL_HRL.HRL_Ref_Taster_vertikal,
    EncoderStartPosition01 := GVL_HRL.HRL_Enc_vertikal_I1,
    EncoderStartPosition02 := GVL_HRL.HRL_Enc_vertikal_I2,
    TOF_TSR_TIME := TIME_TSR,
    AutomaticMode := HRL_OperatingModes.F1
);
HRL_RGB_VertikalUp02 := HRL_Skill_RGB_MoveVerticalBackwards.DO_MovingVerticalRGB_01;
HRL_Skill_RGB_MoveHorizontalForwards(
    ESS := ((GVL.diNotAus_Kanal_A) AND (GVL.diNotAus_Kanal_B)),
    TouchSensor01 := GVL_HRL.HRL_Ref_Taster_horizontal,
    EncoderStartPosition01 := GVL_HRL.HRL_Enc_horizontal_I1,
    EncoderStartPosition02 := GVL_HRL.HRL_Enc_horizontal_I2,
    TOF_Time_TSR := TIME_TSR,
    AutomaticMode := HRL_OperatingModes.F1
);
HRL_RGB_HorizontalForwards01 := HRL_Skill_RGB_MoveHorizontalForwards.DO_MovingHorizontalRGB_01;
HRL_Skill_RGB_MoveHorizontalBackwards(
    ESS := ((GVL.diNotAus_Kanal_A) AND (GVL.diNotAus_Kanal_B)),
    TouchSensor01 := GVL_HRL.HRL_Ref_Taster_horizontal,
    EncoderStartPosition01 := GVL_HRL.HRL_Enc_horizontal_I1,
    EncoderStartPosition02 := GVL_HRL.HRL_Enc_horizontal_I2,
    TOF_Time_TSR := TIME_TSR,
    AutomaticMode := HRL_OperatingModes.F1
);
HRL_RGB_HorizontalBackwards02 := HRL_Skill_RGB_MoveHorizontalBackwards.DO_MovingHorizontalRGB_01;

bAuslagernAktiv := HRL_NMethod_Auslagern.Busy OR (HRL_NMethod_Auslagern.CurrentStep <> 0);;

HRL_ControlOfOutputs(
    F4 := HRL_OperatingModes.F4,
    F1 := HRL_OperatingModes.F1,
    A2 := HRL_OperatingModes.A2,
    A1 := HRL_OperatingModes.A1,
    A6 := HRL_OperatingModes.A6,
    Start := HRL_OperatingModes.Start,

    CB_forwards :=
        (HRL_CB_forwards AND NOT bAuslagernAktiv)
        OR HRL_NMethod_Auslagern.REQ_CB_forwards,

    CB_backwards :=
        (HRL_CB_backwards AND NOT bAuslagernAktiv)
        OR HRL_NMethod_Auslagern.REQ_CB_backwards,

    RGB_Forwards01 :=
        (HRL_RGB_Forwards01 AND NOT bAuslagernAktiv)
        OR HRL_NMethod_Auslagern.REQ_RGB_Forwards,

    RGB_Forwards02 :=
        HRL_RGB_Forwards02 AND NOT bAuslagernAktiv,

    RGB_Backwards01 :=
        (HRL_RGB_Backwards01 AND NOT bAuslagernAktiv)
        OR HRL_NMethod_Auslagern.REQ_RGB_Backwards,

    RGB_Backwards02 :=
        HRL_RGB_Backwards02 AND NOT bAuslagernAktiv,

    RGB_VertikalDown01 :=
        (HRL_RGB_VertikalDown01 AND NOT bAuslagernAktiv)
        OR HRL_NMethod_Auslagern.REQ_RGB_VerticalDown,

    RGB_VertikalDown02 :=
        HRL_RGB_VertikalDown02 AND NOT bAuslagernAktiv,

    RGB_VertikalUp01 :=
        (HRL_RGB_VertikalUp01 AND NOT bAuslagernAktiv)
        OR HRL_NMethod_Auslagern.REQ_RGB_VerticalUp,

    RGB_VertikalUp02 :=
        HRL_RGB_VertikalUp02 AND NOT bAuslagernAktiv,

    RGB_HorizontalForwards01 :=
        (HRL_RGB_HorizontalForwards01 AND NOT bAuslagernAktiv)
        OR HRL_NMethod_Auslagern.REQ_RGB_HorizontalForward,

    RGB_HorizontalForwards02 :=
        HRL_RGB_HorizontalForwards02 AND NOT bAuslagernAktiv,

    RGB_HorizontalBackwards01 :=
        (HRL_RGB_HorizontalBackwards01 AND NOT bAuslagernAktiv)
        OR HRL_NMethod_Auslagern.REQ_RGB_HorizontalBackward,

    RGB_HorizontalBackwards02 :=
        HRL_RGB_HorizontalBackwards02 AND NOT bAuslagernAktiv,

    Init_RGB_Forwards := Init_SRM_MotorForwards,
    Init_RGB_Backwards := Init_SRM_MotorBackwards,
    Init_RGB_VertikalUp := Init_RGB_VerticalUp,
    Init_RGB_VertikalDown := Init_RGB_VerticalDown,
    Init_RGB_HorizontalForwads := Init_RGB_HorizontalForwards,
    Init_RGB_HorizontalBackwards := Init_RGB_HorizontalBackwards
);
IF GVL_Sim.bSimMode THEN

    // Outputs in Simulationsabbild schreiben
    GVL_HRL_Sim.HRL_MOT_Foerderband_vorwaerts :=
        HRL_ControlOfOutputs.ConveyorBeltForward;

    GVL_HRL_Sim.HRL_MOT_Foerderband_rueckwaerts :=
        HRL_ControlOfOutputs.ConveyorBeltBackward;

    GVL_HRL_Sim.HRL_MOT_Ausleger_vorwaerts :=
        HRL_ControlOfOutputs.RGB_Forwards;

    GVL_HRL_Sim.HRL_MOT_Ausleger_rueckwaerts :=
        HRL_ControlOfOutputs.RGB_Backwards;

    GVL_HRL_Sim.HRL_MOT_vertikal_runter :=
        HRL_ControlOfOutputs.RGB_VerticalDown;

    GVL_HRL_Sim.HRL_MOT_vertikal_hoch :=
        HRL_ControlOfOutputs.RGB_VerticalUp;

    GVL_HRL_Sim.HRL_MOT_horizontal_zum_Regal :=
        HRL_ControlOfOutputs.RGB_HorizontalForward;

    GVL_HRL_Sim.HRL_MOT_horizontal_zum_Foerderband :=
        HRL_ControlOfOutputs.RGB_HorizontalBackward;

    GVL_HRL_Sim.HRL_K1_1_Zaehler_Zuruecksetzen :=
        GVL_HRL.HRL_K1_1_Zaehler_Zuruecksetzen;

    GVL_HRL_Sim.HRL_K1_2_Zaehler_Zuruecksetzen :=
        GVL_HRL.HRL_K1_2_Zaehler_Zuruecksetzen;

ELSE

    // Outputs auf reale Hardware schreiben
    GVL_HRL.HRL_MOT_Foerderband_vorwaerts :=
        HRL_ControlOfOutputs.ConveyorBeltForward;

    GVL_HRL.HRL_MOT_Foerderband_rueckwaerts :=
        HRL_ControlOfOutputs.ConveyorBeltBackward;

    GVL_HRL.HRL_MOT_Ausleger_vorwaerts :=
        HRL_ControlOfOutputs.RGB_Forwards;

    GVL_HRL.HRL_MOT_Ausleger_rueckwaerts :=
        HRL_ControlOfOutputs.RGB_Backwards;

    GVL_HRL.HRL_MOT_vertikal_runter :=
        HRL_ControlOfOutputs.RGB_VerticalDown;

    GVL_HRL.HRL_MOT_vertikal_hoch :=
        HRL_ControlOfOutputs.RGB_VerticalUp;

    GVL_HRL.HRL_MOT_horizontal_zum_Regal :=
        HRL_ControlOfOutputs.RGB_HorizontalForward;

    GVL_HRL.HRL_MOT_horizontal_zum_Foerderband :=
        HRL_ControlOfOutputs.RGB_HorizontalBackward;

END_IF;

//GEMMA-Mappings
IF HRL_OperatingModes.A1 THEN
    sCurrentGemmaState := 'HRL_OperatingModes.A1';
ELSIF HRL_OperatingModes.A2 THEN
    sCurrentGemmaState := 'HRL_OperatingModes.A2';
ELSIF HRL_OperatingModes.A5 THEN
    sCurrentGemmaState := 'HRL_OperatingModes.A5';
ELSIF HRL_OperatingModes.A6 THEN
    sCurrentGemmaState := 'HRL_OperatingModes.A6';
ELSIF HRL_OperatingModes.F1 THEN
    sCurrentGemmaState := 'HRL_OperatingModes.F1';
ELSIF HRL_OperatingModes.F4 THEN
    sCurrentGemmaState := 'HRL_OperatingModes.F4';
ELSIF HRL_OperatingModes.D1 THEN
    sCurrentGemmaState := 'HRL_OperatingModes.D1';
ELSIF HRL_OperatingModes.D3 THEN
    sCurrentGemmaState := 'HRL_OperatingModes.D3';
END_IF;

IF NOT HRL_OperatingModes.D2 THEN
    sLastNonFailureGemmaState := sCurrentGemmaState;
END_IF;

rtD2(CLK := HRL_OperatingModes.D2);

IF rtD2.Q THEN
    OPCUA.LastGEMMAStateBeforeFailure := sLastNonFailureGemmaState;
END_IF;

END_PROGRAM

// ---- POUs/Moduls/HRL_Skills/HRL_NMethod_Auslagern.TcPOU
{attribute 'OPC.UA.DA.JobMethod' := 'HRL_NMethod_Auslagern'}
FUNCTION_BLOCK HRL_NMethod_Auslagern
VAR_INPUT
    ESS_OK : BOOL;
    AutomaticMode : BOOL;

    HRL_Enc_horizontal_I1 : UDINT;
    HRL_Enc_horizontal_I2 : UDINT;
    HRL_Enc_vertikal_I1 : UDINT;
    HRL_Enc_vertikal_I2 : UDINT;

    HRL_Ref_Taster_horizontal : BOOL;
    HRL_Ref_Taster_vertikal : BOOL;
    HRL_Ref_Taster_Ausleger_vorne : BOOL;
    HRL_Ref_Taster_Ausleger_hinten : BOOL;

    HRL_LS_innen : BOOL;
    HRL_LS_aussen : BOOL;
END_VAR

VAR_OUTPUT
    REQ_CB_forwards : BOOL;
    REQ_CB_backwards : BOOL;

    REQ_RGB_Forwards : BOOL;
    REQ_RGB_Backwards : BOOL;

    REQ_RGB_VerticalDown : BOOL;
    REQ_RGB_VerticalUp : BOOL;

    REQ_RGB_HorizontalForward : BOOL;
    REQ_RGB_HorizontalBackward : BOOL;

    Busy : BOOL;
    Done : BOOL;
    Error : BOOL;
    ErrorId : UDINT;
    CurrentStep : UDINT;
END_VAR

VAR
    MethodCall_Auslagern : BOOL := FALSE;

    callCounterStart : ULINT := 0;
    callCounterAbort : ULINT := 0;
    callCounterCheckState : ULINT := 0;

    jobRunning : BOOL := FALSE;
    jobFinished : BOOL := FALSE;

    step : UDINT := 0;
    lastStep : UDINT := 0;
    bStepChanged : BOOL := FALSE;

    TargetHorizontalShelf_I1 : UDINT := 0;
    TargetHorizontalShelf_I2 : UDINT := 0;
    TargetVerticalShelf_I1 : UDINT := 0;
    TargetVerticalShelf_I2 : UDINT := 0;

    TargetHorizontalTransfer_I1 : UDINT := 0;
    TargetHorizontalTransfer_I2 : UDINT := 0;
    TargetVerticalTransfer_I1 : UDINT := 0;
    TargetVerticalTransfer_I2 : UDINT := 0;

    ActiveTargetHorizontal_I1 : UDINT := 0;
    ActiveTargetHorizontal_I2 : UDINT := 0;
    ActiveTargetVertical_I1 : UDINT := 0;
    ActiveTargetVertical_I2 : UDINT := 0;

    WatchdogTime : TIME := T#15S;

    cmdHorizontal : BOOL := FALSE;
    cmdVertical : BOOL := FALSE;
    cmdAuslegerForward : BOOL := FALSE;
    cmdAuslegerBackward : BOOL := FALSE;
    cmdConveyorForward : BOOL := FALSE;

    dirHorizontalToRegal : BOOL := FALSE;
    dirVerticalDown : BOOL := FALSE;

    bOppositeCommandError : BOOL := FALSE;
    bAbortRequest : BOOL := FALSE;

    fbHorizontal : AxisControl_Encoder;
    fbVertical : AxisControl_Encoder;
    fbAuslegerForward : AxisControl_MultipleInputSensors;
    fbAuslegerBackward : AxisControl_MultipleInputSensors;
    fbConveyorForward : AxisControl_MultipleInputSensors;

    tonWatchdog : TON;
END_VAR

REQ_CB_forwards := FALSE;
REQ_CB_backwards := FALSE;

REQ_RGB_Forwards := FALSE;
REQ_RGB_Backwards := FALSE;

REQ_RGB_VerticalDown := FALSE;
REQ_RGB_VerticalUp := FALSE;

REQ_RGB_HorizontalForward := FALSE;
REQ_RGB_HorizontalBackward := FALSE;

bOppositeCommandError := FALSE;

bStepChanged := (step <> lastStep);
lastStep := step;

IF bAbortRequest THEN
    cmdHorizontal := FALSE;
    cmdVertical := FALSE;
    cmdAuslegerForward := FALSE;
    cmdAuslegerBackward := FALSE;
    cmdConveyorForward := FALSE;

    MethodCall_Auslagern := FALSE;

    Busy := FALSE;
    Done := FALSE;

    jobRunning := FALSE;
    jobFinished := TRUE;

    // Fehlerstatus bewusst nicht überschreiben
    step := 0;
    bAbortRequest := FALSE;
END_IF;

IF bStepChanged THEN
    tonWatchdog(IN := FALSE, PT := WatchdogTime);
END_IF;

tonWatchdog(
    IN := jobRunning AND (step <> 0) AND (step <> 100) AND (step <> 900),
    PT := WatchdogTime
);

IF tonWatchdog.Q THEN
    Error := TRUE;
    ErrorId := 100;
    step := 900;
END_IF;

IF jobRunning AND NOT ESS_OK THEN
    Error := TRUE;
    ErrorId := 1;
    step := 900;
END_IF;

IF jobRunning AND NOT AutomaticMode THEN
    Error := TRUE;
    ErrorId := 2;
    step := 900;
END_IF;

IF step = 50 THEN
    ActiveTargetHorizontal_I1 := TargetHorizontalTransfer_I1;
    ActiveTargetHorizontal_I2 := TargetHorizontalTransfer_I2;
ELSE
    ActiveTargetHorizontal_I1 := TargetHorizontalShelf_I1;
    ActiveTargetHorizontal_I2 := TargetHorizontalShelf_I2;
END_IF;

IF step = 60 THEN
    ActiveTargetVertical_I1 := TargetVerticalTransfer_I1;
    ActiveTargetVertical_I2 := TargetVerticalTransfer_I2;
ELSE
    ActiveTargetVertical_I1 := TargetVerticalShelf_I1;
    ActiveTargetVertical_I2 := TargetVerticalShelf_I2;
END_IF;

dirHorizontalToRegal := (HRL_Enc_horizontal_I1 < ActiveTargetHorizontal_I1);
dirVerticalDown := (HRL_Enc_vertikal_I1 < ActiveTargetVertical_I1);

fbHorizontal(
    MethodCall := cmdHorizontal,
    EmergencyStopSignal := NOT ESS_OK,
    Direction := dirHorizontalToRegal,
    InitStateDrive_Input := FALSE,
    DI01 := HRL_Ref_Taster_horizontal,
    DI02_EncoderStart01 := HRL_Enc_horizontal_I1,
    DI03_EncoderTarget01 := ActiveTargetHorizontal_I1,
    DI04_EncoderStart02 := HRL_Enc_horizontal_I2,
    DI05_EncoderTarget02 := ActiveTargetHorizontal_I2,
    TouchSensorRelief := FALSE,
    TOF_Time_MotorControl := T#0MS,
    TOF_Time_TouchSensorRelief := T#0MS,
    OperatingMode := AutomaticMode
);

fbVertical(
    MethodCall := cmdVertical,
    EmergencyStopSignal := NOT ESS_OK,
    Direction := dirVerticalDown,
    InitStateDrive_Input := FALSE,
    DI01 := HRL_Ref_Taster_vertikal,
    DI02_EncoderStart01 := HRL_Enc_vertikal_I1,
    DI03_EncoderTarget01 := ActiveTargetVertical_I1,
    DI04_EncoderStart02 := HRL_Enc_vertikal_I2,
    DI05_EncoderTarget02 := ActiveTargetVertical_I2,
    TouchSensorRelief := FALSE,
    TOF_Time_MotorControl := T#0MS,
    TOF_Time_TouchSensorRelief := T#0MS,
    OperatingMode := AutomaticMode
);

fbAuslegerForward(
    MethodCall := cmdAuslegerForward,
    EmergencyStopSignal := NOT ESS_OK,
    Direction := TRUE,
    InitStateDrive_Input := FALSE,
    DI01 := HRL_Ref_Taster_Ausleger_hinten,
    DI02 := HRL_Ref_Taster_Ausleger_vorne,
    TouchSensorRelief := FALSE,
    TOF_Time_MotorControl := T#0MS,
    TOF_Time_TouchSensorRelief := T#0MS,
    OperatingMode := AutomaticMode
);

fbAuslegerBackward(
    MethodCall := cmdAuslegerBackward,
    EmergencyStopSignal := NOT ESS_OK,
    Direction := TRUE,
    InitStateDrive_Input := FALSE,
    DI01 := HRL_Ref_Taster_Ausleger_vorne,
    DI02 := HRL_Ref_Taster_Ausleger_hinten,
    TouchSensorRelief := FALSE,
    TOF_Time_MotorControl := T#0MS,
    TOF_Time_TouchSensorRelief := T#0MS,
    OperatingMode := AutomaticMode
);

fbConveyorForward(
    MethodCall := cmdConveyorForward,
    EmergencyStopSignal := NOT ESS_OK,
    Direction := TRUE,
    InitStateDrive_Input := FALSE,
    DI01 := HRL_LS_innen,
    DI02 := HRL_LS_aussen,
    TouchSensorRelief := FALSE,
    TOF_Time_MotorControl := T#0MS,
    TOF_Time_TouchSensorRelief := T#0MS,
    OperatingMode := AutomaticMode
);

CASE step OF

    0:
        Busy := FALSE;

        cmdHorizontal := FALSE;
        cmdVertical := FALSE;
        cmdAuslegerForward := FALSE;
        cmdAuslegerBackward := FALSE;
        cmdConveyorForward := FALSE;

        jobRunning := FALSE;

        // WICHTIG:
        // Done, Error, ErrorId und jobFinished hier NICHT pauschal löschen.
        // Diese Werte bleiben stehen, bis ein neuer Auftrag startet.

        IF MethodCall_Auslagern THEN

            IF NOT ESS_OK THEN
                Error := TRUE;
                ErrorId := 1;
                MethodCall_Auslagern := FALSE;
                jobFinished := TRUE;
                step := 900;

            ELSIF NOT AutomaticMode THEN
                Error := TRUE;
                ErrorId := 2;
                MethodCall_Auslagern := FALSE;
                jobFinished := TRUE;
                step := 900;

            ELSE
                Done := FALSE;
                Error := FALSE;
                ErrorId := 0;

                Busy := TRUE;
                jobRunning := TRUE;
                jobFinished := FALSE;

                step := 10;
            END_IF;

        END_IF;


    10:
        Busy := TRUE;

        cmdHorizontal := TRUE;
        cmdVertical := FALSE;
        cmdAuslegerForward := FALSE;
        cmdAuslegerBackward := FALSE;
        cmdConveyorForward := FALSE;

        IF dirHorizontalToRegal THEN
            REQ_RGB_HorizontalForward := fbHorizontal.DigitalOutputControl_01;
        ELSE
            REQ_RGB_HorizontalBackward := fbHorizontal.DigitalOutputControl_01;
        END_IF;

        IF REQ_RGB_HorizontalForward AND REQ_RGB_HorizontalBackward THEN
            Error := TRUE;
            ErrorId := 200;
            step := 900;
        END_IF;

        IF fbHorizontal.ResetMethodCall THEN
            cmdHorizontal := FALSE;
            step := 20;
        END_IF;


    20:
        Busy := TRUE;

        cmdHorizontal := FALSE;
        cmdVertical := TRUE;
        cmdAuslegerForward := FALSE;
        cmdAuslegerBackward := FALSE;
        cmdConveyorForward := FALSE;

        IF dirVerticalDown THEN
            REQ_RGB_VerticalDown := fbVertical.DigitalOutputControl_01;
        ELSE
            REQ_RGB_VerticalUp := fbVertical.DigitalOutputControl_01;
        END_IF;

        IF REQ_RGB_VerticalDown AND REQ_RGB_VerticalUp THEN
            Error := TRUE;
            ErrorId := 201;
            step := 900;
        END_IF;

        IF fbVertical.ResetMethodCall THEN
            cmdVertical := FALSE;
            step := 30;
        END_IF;


    30:
        Busy := TRUE;

        cmdHorizontal := FALSE;
        cmdVertical := FALSE;
        cmdAuslegerForward := TRUE;
        cmdAuslegerBackward := FALSE;
        cmdConveyorForward := FALSE;

        REQ_RGB_Forwards := fbAuslegerForward.DigitalOutputControl_01;

        IF REQ_RGB_Forwards AND REQ_RGB_Backwards THEN
            Error := TRUE;
            ErrorId := 202;
            step := 900;
        END_IF;

        IF fbAuslegerForward.ResetMethodCall THEN
            cmdAuslegerForward := FALSE;
            step := 40;
        END_IF;


    40:
        Busy := TRUE;

        cmdHorizontal := FALSE;
        cmdVertical := FALSE;
        cmdAuslegerForward := FALSE;
        cmdAuslegerBackward := TRUE;
        cmdConveyorForward := FALSE;

        REQ_RGB_Backwards := fbAuslegerBackward.DigitalOutputControl_01;

        IF REQ_RGB_Forwards AND REQ_RGB_Backwards THEN
            Error := TRUE;
            ErrorId := 203;
            step := 900;
        END_IF;

        IF fbAuslegerBackward.ResetMethodCall THEN
            cmdAuslegerBackward := FALSE;
            step := 50;
        END_IF;


    50:
        Busy := TRUE;

        cmdHorizontal := TRUE;
        cmdVertical := FALSE;
        cmdAuslegerForward := FALSE;
        cmdAuslegerBackward := FALSE;
        cmdConveyorForward := FALSE;

        IF dirHorizontalToRegal THEN
            REQ_RGB_HorizontalForward := fbHorizontal.DigitalOutputControl_01;
        ELSE
            REQ_RGB_HorizontalBackward := fbHorizontal.DigitalOutputControl_01;
        END_IF;

        IF REQ_RGB_HorizontalForward AND REQ_RGB_HorizontalBackward THEN
            Error := TRUE;
            ErrorId := 204;
            step := 900;
        END_IF;

        IF fbHorizontal.ResetMethodCall THEN
            cmdHorizontal := FALSE;
            step := 60;
        END_IF;


    60:
        Busy := TRUE;

        cmdHorizontal := FALSE;
        cmdVertical := TRUE;
        cmdAuslegerForward := FALSE;
        cmdAuslegerBackward := FALSE;
        cmdConveyorForward := FALSE;

        IF dirVerticalDown THEN
            REQ_RGB_VerticalDown := fbVertical.DigitalOutputControl_01;
        ELSE
            REQ_RGB_VerticalUp := fbVertical.DigitalOutputControl_01;
        END_IF;

        IF REQ_RGB_VerticalDown AND REQ_RGB_VerticalUp THEN
            Error := TRUE;
            ErrorId := 205;
            step := 900;
        END_IF;

        IF fbVertical.ResetMethodCall THEN
            cmdVertical := FALSE;
            step := 65;
        END_IF;


    65:
        Busy := TRUE;

        cmdHorizontal := FALSE;
        cmdVertical := FALSE;
        cmdAuslegerForward := FALSE;
        cmdAuslegerBackward := FALSE;
        cmdConveyorForward := FALSE;

        IF HRL_LS_innen THEN
            step := 70;
        END_IF;


    70:
        Busy := TRUE;

        cmdHorizontal := FALSE;
        cmdVertical := FALSE;
        cmdAuslegerForward := FALSE;
        cmdAuslegerBackward := FALSE;
        cmdConveyorForward := TRUE;

        REQ_CB_forwards := fbConveyorForward.DigitalOutputControl_01;

        IF REQ_CB_forwards AND REQ_CB_backwards THEN
            Error := TRUE;
            ErrorId := 206;
            step := 900;
        END_IF;

        IF fbConveyorForward.ResetMethodCall THEN
            cmdConveyorForward := FALSE;
            step := 100;
        END_IF;


    100:
        REQ_CB_forwards := FALSE;
        REQ_CB_backwards := FALSE;

        REQ_RGB_Forwards := FALSE;
        REQ_RGB_Backwards := FALSE;

        REQ_RGB_VerticalDown := FALSE;
        REQ_RGB_VerticalUp := FALSE;

        REQ_RGB_HorizontalForward := FALSE;
        REQ_RGB_HorizontalBackward := FALSE;

        cmdHorizontal := FALSE;
        cmdVertical := FALSE;
        cmdAuslegerForward := FALSE;
        cmdAuslegerBackward := FALSE;
        cmdConveyorForward := FALSE;

        Busy := FALSE;
        Done := TRUE;
        Error := FALSE;
        ErrorId := 0;

        jobRunning := FALSE;
        jobFinished := TRUE;

        MethodCall_Auslagern := FALSE;

        step := 0;


    900:
        REQ_CB_forwards := FALSE;
        REQ_CB_backwards := FALSE;

        REQ_RGB_Forwards := FALSE;
        REQ_RGB_Backwards := FALSE;

        REQ_RGB_VerticalDown := FALSE;
        REQ_RGB_VerticalUp := FALSE;

        REQ_RGB_HorizontalForward := FALSE;
        REQ_RGB_HorizontalBackward := FALSE;

        cmdHorizontal := FALSE;
        cmdVertical := FALSE;
        cmdAuslegerForward := FALSE;
        cmdAuslegerBackward := FALSE;
        cmdConveyorForward := FALSE;

        Busy := FALSE;
        Done := FALSE;

        jobRunning := FALSE;
        jobFinished := TRUE;

        MethodCall_Auslagern := FALSE;

        // Error und ErrorId absichtlich stehen lassen
        step := 0;

ELSE
    REQ_CB_forwards := FALSE;
    REQ_CB_backwards := FALSE;

    REQ_RGB_Forwards := FALSE;
    REQ_RGB_Backwards := FALSE;

    REQ_RGB_VerticalDown := FALSE;
    REQ_RGB_VerticalUp := FALSE;

    REQ_RGB_HorizontalForward := FALSE;
    REQ_RGB_HorizontalBackward := FALSE;

    cmdHorizontal := FALSE;
    cmdVertical := FALSE;
    cmdAuslegerForward := FALSE;
    cmdAuslegerBackward := FALSE;
    cmdConveyorForward := FALSE;

    Busy := FALSE;
    Done := FALSE;
    Error := TRUE;
    ErrorId := 998;

    jobRunning := FALSE;
    jobFinished := TRUE;

    MethodCall_Auslagern := FALSE;

    step := 0;
END_CASE;

CurrentStep := step;

{attribute 'TcRpcEnable' := '1'}
METHOD Abort : HRESULT
VAR_INPUT
    hdl : UDINT;
END_VAR
callCounterAbort := callCounterAbort + 1;

bAbortRequest := TRUE;

Abort := 0;
END_METHOD

{attribute 'TcRpcEnable' := '1'}
METHOD CheckState : HRESULT
VAR_INPUT
    hdl : UDINT;
END_VAR

VAR_OUTPUT
    bBusy : BOOL;
    State : UDINT;
    IsDone : BOOL;
    HasError : BOOL;
    ErrorCode : UDINT;
END_VAR
callCounterCheckState := callCounterCheckState + 1;

bBusy := jobRunning;
State := CurrentStep;
IsDone := jobFinished;
HasError := Error;
ErrorCode := ErrorId;

CheckState := 0;
END_METHOD

{attribute 'TcRpcEnable' := '1'}
METHOD Start : HRESULT
VAR_INPUT
    MethodCall : BOOL;

    HorizontalShelf_I1 : UDINT;
    HorizontalShelf_I2 : UDINT;
    VerticalShelf_I1 : UDINT;
    VerticalShelf_I2 : UDINT;

    HorizontalTransfer_I1 : UDINT;
    HorizontalTransfer_I2 : UDINT;
    VerticalTransfer_I1 : UDINT;
    VerticalTransfer_I2 : UDINT;

    Timeout : TIME;
END_VAR

VAR_OUTPUT
    hdl : UDINT;
END_VAR
callCounterStart := callCounterStart + 1;

IF NOT jobRunning THEN
	 IF MethodCall THEN
        OPCUA.lastExecutedProcess := 'HRL_NMethod_Auslagern';
        OPCUA.lastExecutedSkill := 'HRL_NMethod_Auslagern';
    END_IF;
    MethodCall_Auslagern := MethodCall;

    TargetHorizontalShelf_I1 := HorizontalShelf_I1;
    TargetHorizontalShelf_I2 := HorizontalShelf_I2;
    TargetVerticalShelf_I1 := VerticalShelf_I1;
    TargetVerticalShelf_I2 := VerticalShelf_I2;

    TargetHorizontalTransfer_I1 := HorizontalTransfer_I1;
    TargetHorizontalTransfer_I2 := HorizontalTransfer_I2;
    TargetVerticalTransfer_I1 := VerticalTransfer_I1;
    TargetVerticalTransfer_I2 := VerticalTransfer_I2;

    IF Timeout > T#0MS THEN
        WatchdogTime := Timeout;
    ELSE
        WatchdogTime := T#15S;
    END_IF;

    // Neuer Auftrag löscht alten Abschlussstatus
    jobFinished := FALSE;
    Done := FALSE;
    Error := FALSE;
    ErrorId := 0;

    hdl := 1;
    Start := 0;
ELSE
    hdl := 0;
    Start := 16#800700AA;
END_IF;
END_METHOD

END_FUNCTION_BLOCK

// ---- POUs/AtomicSkillsSchablonen/AxisControl_Encoder.TcPOU
FUNCTION_BLOCK AxisControl_Encoder
VAR_INPUT //Input-Variablen des FBs
	MethodCall					: BOOL; // Variable zum aktiven Aufruf einer OPC UA Methode
	EmergencyStopSignal 		: BOOL; // Variable für Not-Signal 
	Direction 					: BOOL; // Variable zur Bestimmung der Bewegungsrichtung
	InitStateDrive_Input		: BOOL; //InputVariable für Initialfahrt
	DI01 						: BOOL; // Digitaler Input wie bspw. Lichtsensor oder Kontaktsensor 
	DI02_EncoderStart01			: UDINT; // Digitaler Input Encoder Wert
	DI03_EncoderTarget01		: UDINT; // Digitaler Input Encoder Wert
	DI04_EncoderStart02			: UDINT; // Digitaler Input Encoder Wert
	DI05_EncoderTarget02		: UDINT; // Digitaler Input Encoder Wert
	TouchSensorRelief 			: BOOL; // Hilfsvariable zur Identifikation ob eine Endschalterentlastung notwendig ist
	TOF_Time_MotorControl		: TIME; // Zeitvariable für die Ausschaltverzögerung des digitalen Outputs (Motoransteuerung) 
	TOF_Time_TouchSensorRelief	: TIME; // Ausschaltverzögerung für die Endschaltentlastung
	OperatingMode				: BOOL; // Variable zur Festlegung des benötigten Betriebszustandes für die Auslösung des FBs
END_VAR

VAR_OUTPUT //Output-Variablen des FBs
	DigitalOutputControl_01	: BOOL; //Digitale Output Ansteuerung des Motor 1
	DigitalOutputControl_02	: BOOL; //Digitale Output Ansteuerung des Motor 2
	ResetMethodCall			: BOOL; //Outputvariable für den Reset der OPC UA Methode
END_VAR

VAR //Interne-Variablen des FBs
//FlipFlop
	RS_AxisControl		: RS; //FlipFlop für die Ansteuerung der Achse oder des Transportbandes
	RS_TouchSensorRelief: RS; //FlipFlop zu Ansteuerung der Endschalterentlastung
//Zeitverzögerung
	TOF_TouchSensorRelief	: TOF; //Ausschaltverzögerung für die Endschalterentlastung
	TOF_DigitalOutputControl: TOF; //Ausschaltverzögerung für die Outputansteuerung
//Flanke	
	R_TRIG_MethodCall			: R_TRIG; //Flankenerkennung für eingehenden MethodenCall
	R_TRIG_EncoderPos01_Input	: R_TRIG; //Flankenerkennung für Vergleich der Encoderwerte von Start- und Zielposition
	R_TRIG_EncoderPos02_Input	: R_TRIG; //Flankenerkennung für Vergleich der Encoderwerte von Start- und Zielposition
	R_TRIG_EncoderPos01_Output	: R_TRIG; //Flankenerkennung für Vergleich der Encoderwerte von Start- und Zielposition
	R_TRIG_EncoderPos02_Output	: R_TRIG; //Flankenerkennung für Vergleich der Encoderwerte von Start- und Zielposition
END_VAR

R_TRIG_MethodCall(CLK := MethodCall);

ResetMethodCall := (
    (Direction AND (DI02_EncoderStart01 >= DI03_EncoderTarget01) AND (DI04_EncoderStart02 >= DI05_EncoderTarget02))
    OR ((NOT Direction) AND (DI02_EncoderStart01 <= DI03_EncoderTarget01) AND (DI04_EncoderStart02 <= DI05_EncoderTarget02))
    OR EmergencyStopSignal
    OR DI01
    OR InitStateDrive_Input
);

RS_AxisControl(
    SET := (
        R_TRIG_MethodCall.Q
        AND (
            (Direction AND (DI02_EncoderStart01 < DI03_EncoderTarget01) AND (DI04_EncoderStart02 < DI05_EncoderTarget02))
            OR ((NOT Direction) AND (DI02_EncoderStart01 > DI03_EncoderTarget01) AND (DI04_EncoderStart02 > DI05_EncoderTarget02))
            OR InitStateDrive_Input
        )
        AND OperatingMode
    ),
    RESET1 := ResetMethodCall
);

TOF_DigitalOutputControl(IN := RS_AxisControl.Q1, PT := TOF_Time_MotorControl);
DigitalOutputControl_01 := TOF_DigitalOutputControl.Q;

RS_TouchSensorRelief(
    SET := ((ResetMethodCall) AND (MethodCall) AND (TouchSensorRelief)),
    RESET1 := ((NOT DI01) OR EmergencyStopSignal OR InitStateDrive_Input)
);
TOF_TouchSensorRelief(IN := RS_TouchSensorRelief.Q1, PT := TOF_Time_TouchSensorRelief);
DigitalOutputControl_02 := TOF_TouchSensorRelief.Q;

END_FUNCTION_BLOCK

// ---- POUs/AtomicSkillsSchablonen/AxisControl_MultipleInputSensors.TcPOU
FUNCTION_BLOCK AxisControl_MultipleInputSensors
VAR_INPUT//Input-Variablen des FBs
	MethodCall					: BOOL; // Variable zum aktiven Aufruf einer OPC UA Methode
	EmergencyStopSignal 		: BOOL; // Variable für Not-Signal 
	Direction 					: BOOL; // Variable zur Bestimmung der Bewegungsrichtung
	InitStateDrive_Input		: BOOL; //InputVariable für Initialfahrt
	DI01 						: BOOL; // Digitaler Input wie bspw. Lichtsensor oder Kontaktsensor 
	DI02 						: BOOL; // Digitaler Input wie bspw. Lichtsensor oder Kontaktsensor 
	TouchSensorRelief			: BOOL; // Hilfsvariable zur Identifikation ob eine Endschalterentlastung notwendig ist
	TOF_Time_MotorControl		: TIME; // Zeitvariable für die Ausschaltverzögerung des digitalen Outputs (Motoransteuerung) 
	TOF_Time_TouchSensorRelief	: TIME; // Ausschaltverzögerung für die Endschaltentlastung
	OperatingMode				: BOOL; // Variable zur Festlegung des benötigten Betriebszustandes für die Auslösung des FBs
END_VAR

VAR_OUTPUT //Output-Variablen des FBs
	DigitalOutputControl_01	: BOOL; //Digitale Output Ansteuerung des Motor 1
	DigitalOutputControl_02	: BOOL; //Digitale Output Ansteuerung des Motor 2
	ResetMethodCall			: BOOL; //Outputvariable für den Reset der OPC UA Methode
	InitStateDriveFinished	: BOOL;
	Count1 : INT := 0;
	Count2 : INT := 0;
END_VAR

VAR //Interne-Variablen des FBs
//FlipFlop
	RS_AxisControl		: RS; //FlipFlop für die Ansteuerung der Achse oder des Transportbandes
	RS_TouchSensorRelief: RS; //FlipFlop zu Ansteuerung der Endschalterentlastung
//Zeitverzögerung
	TOF_TouchSensorRelief	: TOF; //Ausschaltverzögerung für die Endschalterentlastung
	TOF_DigitalOutputControl: TOF; //Ausschaltverzögerung für die Outputansteuerung	
//Flanke	
	R_TRIG_MethodCall : R_TRIG; //Flankenerkennung für eingehenden MethodenCall
	R_TRIG_TSR : R_TRIG; //Flankenerkennung für eingehenden MethodenCall
	F_TRIG_0: F_TRIG;
	F_TRIG_1: F_TRIG;
END_VAR

R_TRIG_MethodCall(CLK := MethodCall);
ResetMethodCall := ((((Direction) AND (DI02))) OR (EmergencyStopSignal));
RS_AxisControl(
    SET := ((R_TRIG_MethodCall.Q) AND (((((Direction) AND (((DI01) OR (TouchSensorRelief))))) OR (((Direction) AND (InitStateDrive_Input))))) AND (OperatingMode)),
    RESET1 := ((((Direction) AND (DI02))) OR (EmergencyStopSignal))
);
TOF_DigitalOutputControl(IN := RS_AxisControl.Q1, PT := TOF_Time_MotorControl);
DigitalOutputControl_01 := TOF_DigitalOutputControl.Q;
R_TRIG_TSR(CLK := ((ResetMethodCall) AND (DI02) AND (MethodCall) AND (TouchSensorRelief)));
InitStateDriveFinished := ((NOT (DI02)) OR (EmergencyStopSignal));
RS_TouchSensorRelief(SET := R_TRIG_TSR.Q, RESET1 := ((NOT (DI02)) OR (EmergencyStopSignal)));
TOF_TouchSensorRelief(IN := RS_TouchSensorRelief.Q1, PT := TOF_Time_TouchSensorRelief);
DigitalOutputControl_02 := TOF_TouchSensorRelief.Q;
F_TRIG_0(CLK := DigitalOutputControl_01);
F_TRIG_1(CLK := DigitalOutputControl_02);

END_FUNCTION_BLOCK

// ---- POUs/Moduls/HRL_Skills/HRL_CB_AS_HorizontalMoveSensors.TcPOU
{attribute 'OPC.UA.DA.JobMethod' := 'JobMethode_HorizontalMove'}
FUNCTION_BLOCK HRL_CB_AS_HorizontalMoveSensors
VAR
	AlwaysTrue : BOOL := TRUE;
	// Used for debugging purposes to display InputArguments of method call
	MethodCall_HorizontalMove : BOOL := FALSE; // used to store InputArg "MethodCall" from Start() method
	ResetMethodCall	: BOOL := FALSE;
	DirectionHorizontal : BOOL; // defines movement direction
	callCounterStart : ULINT; // counts how many times the Start() method has been called
	callCounterCheckState : ULINT; // counts how many times the CheckState() method has been called
	callCounterAbort : ULINT; // counts how many times the Abort() method has been called
	
	// Variables to determine if a job has been started (Start() method has been called) or finished
	jobRunning : BOOL;
	jobFinished : BOOL;

	// State machine variable
	state : UDINT;
	
	// FB Intatziation Variable
	HRL_CB_HorizontalMove : AxisControl_MultipleInputSensors;
END_VAR
	
VAR_INPUT
	ESS						: BOOL;
	LightBarrierSensor_01 	: BOOL;
	LightBarrierSensor_02 	: BOOL;
	AutomaticMode			: BOOL;
END_VAR

VAR_OUTPUT
	DO_MovingConveyorBelt : BOOL;
END_VAR

HRL_CB_HorizontalMove(
    MethodCall := MethodCall_HorizontalMove,
    EmergencyStopSignal := ESS,
    Direction := DirectionHorizontal,
    InitStateDrive_Input := FALSE,
    DI01 := LightBarrierSensor_01,
    DI02 := LightBarrierSensor_02,
    TouchSensorRelief := FALSE,
    TOF_Time_MotorControl := T#0MS,
    TOF_Time_TouchSensorRelief := T#0MS,
    OperatingMode := AutomaticMode
);
DO_MovingConveyorBelt := HRL_CB_HorizontalMove.DigitalOutputControl_01;

{attribute 'TcRpcEnable' := '1'}
METHOD Abort : HRESULT
VAR_INPUT
	hdl : UDINT; // Do not change, used by server.
END_VAR
callCounterAbort := callCounterAbort + 1;
END_METHOD

{attribute 'TcRpcEnable' := '1'}
METHOD CheckState : HRESULT
VAR_INPUT
	hdl : UDINT; // Do not change, used by server.
END_VAR
VAR_OUTPUT
	bBusy : BOOL; // Do not change. Used by server to find out if the job is finished
	
	// List of OutputArguments for OPC UA method, may be customized
	State : BOOL; // Abgeschlossener MethodCall
	MethodCall: BOOL; //Input Recall
END_VAR
callCounterCheckState := callCounterCheckState + 1;
IF NOT jobFinished THEN
	bBusy := TRUE; // job is not finished yet
	CheckState := 0; // no error
ELSE
	bBusy := FALSE; // job is finished
	CheckState := 0; // done, no error occured during execution (OPC UA StatusCode "GOOD")
	jobFinished := FALSE;
	State := ResetMethodCall;
	MethodCall := MethodCall_HorizontalMove;
END_IF
END_METHOD

{attribute 'TcRpcEnable' := '1'}
METHOD Start : HRESULT
VAR_INPUT
	// List of InputArguments for OPC UA method, may be customized
	MethodCall : BOOL; // some description
	MovementDirection : BOOL;	
END_VAR
VAR_OUTPUT
	hdl : UDINT; // Do not change, used by server.
END_VAR
callCounterStart := callCounterStart + 1;

MethodCall_HorizontalMove := MethodCall;
DirectionHorizontal := MovementDirection;

jobRunning := TRUE;
Start := 0; // no error occured, e.g. while parsing the input arguments (0 = OPC UA StatusCode "GOOD")
END_METHOD

END_FUNCTION_BLOCK

// ---- POUs/Moduls/HRL_Skills/HRL_RGB_AS_HorizontalMoveSensors.TcPOU
{attribute 'OPC.UA.DA.JobMethod' := 'JobMethode_HorizontalMove'}
FUNCTION_BLOCK HRL_RGB_AS_HorizontalMoveSensors
VAR
	AlwaysTrue : BOOL := TRUE;
	// Used for debugging purposes to display InputArguments of method call
	MethodCall_HorizontalMove : BOOL := FALSE; // used to store InputArg "MethodCall" from Start() method
	ResetMethodCall	: BOOL := FALSE;	
	DirectionHorizontal : BOOL; // defines movement direction
	TSR : BOOL; // Variable that is needed to perform the relief of the touch sensor
	callCounterStart : ULINT; // counts how many times the Start() method has been called
	callCounterCheckState : ULINT; // counts how many times the CheckState() method has been called
	callCounterAbort : ULINT; // counts how many times the Abort() method has been called
	
	// Variables to determine if a job has been started (Start() method has been called) or finished
	jobRunning : BOOL;
	jobFinished : BOOL;

	// State machine variable
	state : UDINT;
	
	// FB Intatziation Variable
	HRL_RGB_HorizontalMove : AxisControl_MultipleInputSensors;
END_VAR
	
VAR_INPUT
	ESS				: BOOL;
	TouchSensor01 	: BOOL;
	TouchSensor02 	: BOOL;
	TOF_Time_TSR 	: TIME;
	AutomaticMode	: BOOL;
END_VAR

VAR_OUTPUT
	DO_MovingHorizontalRGB_01 : BOOL;
	DO_MovingHorizontalRGB_02 : BOOL;
END_VAR

HRL_RGB_HorizontalMove(
    MethodCall := MethodCall_HorizontalMove,
    EmergencyStopSignal := ESS,
    Direction := DirectionHorizontal,
    InitStateDrive_Input := FALSE,
    DI01 := TouchSensor01,
    DI02 := TouchSensor02,
    TouchSensorRelief := TSR,
    TOF_Time_MotorControl := T#0MS,
    TOF_Time_TouchSensorRelief := TOF_Time_TSR,
    OperatingMode := AutomaticMode
);
DO_MovingHorizontalRGB_01 := HRL_RGB_HorizontalMove.DigitalOutputControl_01;

{attribute 'TcRpcEnable' := '1'}
METHOD Abort : HRESULT
VAR_INPUT
	hdl : UDINT; // Do not change, used by server.
END_VAR
callCounterAbort := callCounterAbort + 1;
END_METHOD

{attribute 'TcRpcEnable' := '1'}
METHOD CheckState : HRESULT
VAR_INPUT
	hdl : UDINT; // Do not change, used by server.
END_VAR
VAR_OUTPUT
	bBusy : BOOL; // Do not change. Used by server to find out if the job is finished
	
	// List of OutputArguments for OPC UA method, may be customized
	State : BOOL; // Abgeschlossener MethodCall
	MethodCall: BOOL; //Input Recall
END_VAR
callCounterCheckState := callCounterCheckState + 1;
IF NOT jobFinished THEN
	bBusy := TRUE; // job is not finished yet
	CheckState := 0; // no error
ELSE
	bBusy := FALSE; // job is finished
	CheckState := 0; // done, no error occured during execution (OPC UA StatusCode "GOOD")
	jobFinished := FALSE;
	State := ResetMethodCall;
	MethodCall := MethodCall_HorizontalMove;
END_IF
END_METHOD

{attribute 'TcRpcEnable' := '1'}
METHOD Start : HRESULT
VAR_INPUT
	// List of InputArguments for OPC UA method, may be customized
	MethodCall : BOOL; // some description
	MovementDirection : BOOL;
	TouchSensorRelief : BOOL;
END_VAR
VAR_OUTPUT
	hdl : UDINT; // Do not change, used by server.
END_VAR
callCounterStart := callCounterStart + 1;

MethodCall_HorizontalMove := MethodCall;
DirectionHorizontal := MovementDirection;
TSR := TouchSensorRelief;

jobRunning := TRUE;
Start := 0; // OPC UA StatusCode GOOD
END_METHOD

END_FUNCTION_BLOCK

// ---- POUs/Moduls/HRL_Skills/HRL_RGB_AS_VerticalMoveEncoders.TcPOU
{attribute 'OPC.UA.DA.JobMethod' := 'JobMethode_VerticalMove'}
FUNCTION_BLOCK HRL_RGB_AS_VerticalMoveEncoders
VAR
	AlwaysTrue : BOOL := TRUE;
	// Used for debugging purposes to display InputArguments of method call
	MethodCall_VerticalMove : BOOL := FALSE; // used to store InputArg "MethodCall" from Start() method
	ResetMethodCall	: BOOL := FALSE;
	DirectionVertical : BOOL;
	EncoderTargetPosition01 : UDINT;
	EncoderTargetPosition02 : UDINT;
	TSR : BOOL;
	callCounterStart : ULINT; // counts how many times the Start() method has been called
	callCounterCheckState : ULINT; // counts how many times the CheckState() method has been called
	callCounterAbort : ULINT; // counts how many times the Abort() method has been called
	
	// Variables to determine if a job has been started (Start() method has been called) or finished
	jobRunning : BOOL;
	jobFinished : BOOL;

	// State machine variable
	state : UDINT;
	
	// FB Intatziation Variable
	HRL_RGB_VerticalMoveWithEncoder : AxisControl_Encoder;
END_VAR
	
VAR_INPUT
	ESS: BOOL;
	TouchSensor01 : BOOL;
	EncoderStartPosition01 : UDINT;
	EncoderStartPosition02 : UDINT;
	TOF_TSR_TIME : TIME;
	AutomaticMode: BOOL;
END_VAR

VAR_OUTPUT
	DO_MovingVerticalRGB_01 : BOOL;
	DO_MovingVerticalRGB_02 : BOOL;
END_VAR

HRL_RGB_VerticalMoveWithEncoder(
    MethodCall := MethodCall_VerticalMove,
    EmergencyStopSignal := ESS,
    Direction := DirectionVertical,
    InitStateDrive_Input := FALSE,
    DI01 := TouchSensor01,
    DI02_EncoderStart01 := EncoderStartPosition01,
    DI03_EncoderTarget01 := EncoderTargetPosition01,
    DI04_EncoderStart02 := EncoderStartPosition02,
    DI05_EncoderTarget02 := EncoderTargetPosition02,
    TouchSensorRelief := TSR,
    TOF_Time_MotorControl := T#0MS,
    TOF_Time_TouchSensorRelief := TOF_TSR_TIME,
    OperatingMode := AutomaticMode
);
DO_MovingVerticalRGB_01 := HRL_RGB_VerticalMoveWithEncoder.DigitalOutputControl_01;

{attribute 'TcRpcEnable' := '1'}
METHOD Abort : HRESULT
VAR_INPUT
	hdl : UDINT; // Do not change, used by server.
END_VAR
callCounterAbort := callCounterAbort + 1;
END_METHOD

{attribute 'TcRpcEnable' := '1'}
METHOD CheckState : HRESULT
VAR_INPUT
	hdl : UDINT; // Do not change, used by server.
END_VAR
VAR_OUTPUT
	bBusy : BOOL; // Do not change. Used by server to find out if the job is finished
	
	// List of OutputArguments for OPC UA method, may be customized
	State : BOOL; // Abgeschlossener MethodCall
	MethodCall: BOOL; //Input Recall
END_VAR
callCounterCheckState := callCounterCheckState + 1;
IF NOT jobFinished THEN
	bBusy := TRUE; // job is not finished yet
	CheckState := 0; // no error
ELSE
	bBusy := FALSE; // job is finished
	CheckState := 0; // done, no error occured during execution (OPC UA StatusCode "GOOD")
	jobFinished := FALSE;
	State := ResetMethodCall;
	MethodCall := MethodCall_VerticalMove;
END_IF
END_METHOD

{attribute 'TcRpcEnable' := '1'}
METHOD Start : HRESULT
VAR_INPUT
	// List of InputArguments for OPC UA method, may be customized
	MethodCall : BOOL; // some description
	MovementDirection : BOOL;
	EncoderPositionVertical_01 : UDINT;
	EncoderPositionVertical_02 : UDINT;
	TouchSensorRelief : BOOL;
END_VAR
VAR_OUTPUT
	hdl : UDINT; // Do not change, used by server.
END_VAR
callCounterStart := callCounterStart + 1;

MethodCall_VerticalMove := MethodCall;
DirectionVertical := MovementDirection;
EncoderTargetPosition01 := EncoderPositionVertical_01;
EncoderTargetPosition02 := EncoderPositionVertical_02;
TSR := TouchSensorRelief;

jobRunning := TRUE;
Start := 0; // no error occured, e.g. while parsing the input arguments (0 = OPC UA StatusCode "GOOD")
END_METHOD

END_FUNCTION_BLOCK

// ---- POUs/Moduls/HRL_Skills/HRL_RGB_AS_HorizontalMoveEncoders.TcPOU
{attribute 'OPC.UA.DA.JobMethod' := 'JobMethode_HorizontalMove'}
FUNCTION_BLOCK HRL_RGB_AS_HorizontalMoveEncoders
VAR
	AlwaysTrue : BOOL := TRUE;
	// Used for debugging purposes to display InputArguments of method call
	MethodCall_HorizontalMove : BOOL := FALSE; // used to store InputArg "MethodCall" from Start() method
	ResetMethodCall	: BOOL := FALSE;	
	DirectionHorizontal : BOOL;
	EncoderTargetPosition01 : UDINT;
	EncoderTargetPosition02 : UDINT;
	TSR: BOOL;
	callCounterStart : ULINT; // counts how many times the Start() method has been called
	callCounterCheckState : ULINT; // counts how many times the CheckState() method has been called
	callCounterAbort : ULINT; // counts how many times the Abort() method has been called
	
	// Variables to determine if a job has been started (Start() method has been called) or finished
	jobRunning : BOOL;
	jobFinished : BOOL;

	// State machine variable
	state : UDINT;
	
	// FB Intatziation Variable
	HRL_RGB_HorizontalMoveWithEncoder : AxisControl_Encoder;
END_VAR
	
VAR_INPUT
	ESS						: BOOL;
	TouchSensor01 			: BOOL;
	EncoderStartPosition01 	: UDINT;
	EncoderStartPosition02 	: UDINT;
	TOF_Time_TSR 			: TIME;
	AutomaticMode			: BOOL;
END_VAR

VAR_OUTPUT
	DO_MovingHorizontalRGB_01 : BOOL;
	DO_MovingHorizontalRGB_02 : BOOL;
END_VAR

HRL_RGB_HorizontalMoveWithEncoder(
    MethodCall := MethodCall_HorizontalMove,
    EmergencyStopSignal := ESS,
    Direction := DirectionHorizontal,
    InitStateDrive_Input := FALSE,
    DI01 := TouchSensor01,
    DI02_EncoderStart01 := EncoderStartPosition01,
    DI03_EncoderTarget01 := EncoderTargetPosition01,
    DI04_EncoderStart02 := EncoderStartPosition02,
    DI05_EncoderTarget02 := EncoderTargetPosition02,
    TouchSensorRelief := TSR,
    TOF_Time_MotorControl := T#0MS,
    TOF_Time_TouchSensorRelief := TOF_Time_TSR,
    OperatingMode := AutomaticMode
);
DO_MovingHorizontalRGB_01 := HRL_RGB_HorizontalMoveWithEncoder.DigitalOutputControl_01;

{attribute 'TcRpcEnable' := '1'}
METHOD Abort : HRESULT
VAR_INPUT
	hdl : UDINT; // Do not change, used by server.
END_VAR
callCounterAbort := callCounterAbort + 1;
END_METHOD

{attribute 'TcRpcEnable' := '1'}
METHOD CheckState : HRESULT
VAR_INPUT
	hdl : UDINT; // Do not change, used by server.
END_VAR
VAR_OUTPUT
	bBusy : BOOL; // Do not change. Used by server to find out if the job is finished
	
	// List of OutputArguments for OPC UA method, may be customized
	State : BOOL; // Abgeschlossener MethodCall
	MethodCall: BOOL; //Input Recall
END_VAR
callCounterCheckState := callCounterCheckState + 1;
IF NOT jobFinished THEN
	bBusy := TRUE; // job is not finished yet
	CheckState := 0; // no error
ELSE
	bBusy := FALSE; // job is finished
	CheckState := 0; // done, no error occured during execution (OPC UA StatusCode "GOOD")
	jobFinished := FALSE;
	State := ResetMethodCall;
	MethodCall := MethodCall_HorizontalMove;
END_IF
END_METHOD

{attribute 'TcRpcEnable' := '1'}
METHOD Start : HRESULT
VAR_INPUT
	// List of InputArguments for OPC UA method, may be customized
	MethodCall : BOOL; // some description
	MovementDirection : BOOL;
	EncoderPositionHorizontal_01 : UDINT;
	EncoderPositionHorizontal_02 : UDINT;
	TouchSensorRelief : BOOL;
END_VAR
VAR_OUTPUT
	hdl : UDINT; // Do not change, used by server.
END_VAR
callCounterStart := callCounterStart + 1;

MethodCall_HorizontalMove := MethodCall;
DirectionHorizontal := MovementDirection;
EncoderTargetPosition01 := EncoderPositionHorizontal_01;
EncoderTargetPosition02 := EncoderPositionHorizontal_02;
TSR := TouchSensorRelief;

jobRunning := TRUE;
Start := 0; // no error occured, e.g. while parsing the input arguments (0 = OPC UA StatusCode "GOOD")
END_METHOD

END_FUNCTION_BLOCK

// ---- POUs/ControlOfOutputs/HRL_ControlOfOutputs.TcPOU
FUNCTION_BLOCK HRL_ControlOfOutputs
VAR_INPUT
	F4							: BOOL;
	F1							: BOOL;
	A2							: BOOL;
	A6							: BOOL;
	A1							: BOOL := FALSE;
	Start						: BOOL;
	CB_forwards 				: BOOL; 
	CB_backwards 				: BOOL; 
	RGB_Forwards01 				: BOOL;
	RGB_Forwards02 				: BOOL;
	RGB_Backwards01				: BOOL; 
	RGB_Backwards02 			: BOOL; 
	RGB_VertikalDown01			: BOOL; 
	RGB_VertikalDown02			: BOOL; 
	RGB_VertikalUp01			: BOOL;
	RGB_VertikalUp02			: BOOL; 
	RGB_HorizontalForwards01 	: BOOL; 
	RGB_HorizontalForwards02	: BOOL;
	RGB_HorizontalBackwards01 	: BOOL; 
	RGB_HorizontalBackwards02 	: BOOL;
	Init_RGB_Forwards			: BOOL;
	Init_RGB_Backwards			: BOOL;
	Init_RGB_VertikalUp			: BOOL;
	Init_RGB_VertikalDown		: BOOL;
	Init_RGB_HorizontalForwads 	: BOOL;
	Init_RGB_HorizontalBackwards : BOOL;
END_VAR
VAR_OUTPUT
	ConveyorBeltForward: BOOL;
	ConveyorBeltBackward: BOOL;
	RGB_Forwards: BOOL;
	RGB_Backwards: BOOL;
	RGB_VerticalDown: BOOL;
	RGB_VerticalUp: BOOL;
	RGB_HorizontalForward: BOOL;
	RGB_HorizontalBackward: BOOL;
	Light_Q1: BOOL;
	Light_Q2: BOOL;
	Light_Q3: BOOL;
END_VAR
VAR
END_VAR

 ConveyorBeltForward := ((((((F1) OR (A2))) AND (CB_Forwards))) OR (((Start) AND (F4))));
ConveyorBeltBackward := ((((((F1) OR (A2))) AND (CB_Backwards))) OR (((Start) AND (F4))));
RGB_Forwards := ((((((F1) OR (A2))) AND (((RGB_Forwards01) OR (RGB_Forwards02))))) OR (((Start) AND (F4))) OR (((A6) AND (Init_RGB_Forwards))));
RGB_Backwards := ((((((F1) OR (A2))) AND (((RGB_Backwards01) OR (RGB_Backwards02))))) OR (((Start) AND (F4))) OR (((A6) AND (Init_RGB_Backwards))));
RGB_VerticalDown := ((((((F1) OR (A2))) AND (((RGB_VertikalDown01) OR (RGB_VertikalDown02))))) OR (((Start) AND (F4))) OR (((A6) AND (Init_RGB_VertikalDown))));
RGB_VerticalUp := ((((((F1) OR (A2))) AND (((RGB_VertikalUp01) OR (RGB_VertikalUp02))))) OR (((Start) AND (F4))) OR (((A6) AND (Init_RGB_VertikalUp))));
RGB_HorizontalForward := ((((((F1) OR (A2))) AND (((RGB_HorizontalForwards01) OR (RGB_HorizontalForwards02))))) OR (((Start) AND (F4))) OR (((A6) AND (Init_RGB_HorizontalForwads))));
RGB_HorizontalBackward := ((((((F1) OR (A2))) AND (((RGB_HorizontalBackwards01) OR (RGB_HorizontalBackwards02))))) OR (((Start) AND (F4))) OR (((A6) AND (Init_RGB_HorizontalBackwards))));
Light_Q1 := F1;
Light_Q2 := F4;
Light_Q3 := A1;

END_FUNCTION_BLOCK

// ---- POUs/OperatingModes/HRL_OperatingModes.TcPOU
FUNCTION_BLOCK HRL_OperatingModes
VAR_INPUT
	Start 			: BOOL;
	Stop			: BOOL;
	Reset			: BOOL;
	Schalter		: BOOL;
	Schrittkette_GS	: BOOL;
	Count1 : INT := 0;
	Count2 : INT := 0;
	Alt_abort: BOOL;
	Err_detected: BOOL;
	Diag_finished: BOOL;
	Alt_found: BOOL;
	Cycle_finished: BOOL;

END_VAR
VAR_OUTPUT
	{attribute 'OPC.UA.DA' := '1'} // für OPC UA freigeben
	A1 : BOOL := FALSE; //Initialzustand
	{attribute 'OPC.UA.DA' := '1'} // für OPC UA freigeben
	A2 : BOOL; //Stillstand angefordert am Ende des Zyklus
//	A3 : BOOL; //Stillstand angefordert in einem bestimmten Zustand
//	A4 : BOOL; //Erhaltener Stillstand
	{attribute 'OPC.UA.DA' := '1'} // für OPC UA freigeben
	A5 : BOOL; //Vorbereitung zur Wiederaufnahme nach Störung
	{attribute 'OPC.UA.DA' := '1'} // für OPC UA freigeben
	A6 : BOOL; //Fahrt in den Initialzustand
	{attribute 'OPC.UA.DA' := '1'} // für OPC UA freigeben
	F1 : BOOL; //Normalbetrieb
//	F2 : BOOL; //Anfahren
//	F3 : BOOL; //Abfahren
	{attribute 'OPC.UA.DA' := '1'} // für OPC UA freigeben
	F4 : BOOL; //Handbetrieb
//	F5 : BOOL; //Schrittbetrieb
//	F6 : BOOL; //Testbetrieb
	{attribute 'OPC.UA.DA' := '1'} // für OPC UA freigeben
	D1 : BOOL; //Not-Aus
	{attribute 'OPC.UA.DA' := '1'} // für OPC UA freigeben
	D2 : BOOL; //Diagnose und Störbehandlung
	{attribute 'OPC.UA.DA' := '1'} // für OPC UA freigeben
	D3 : BOOL; //Produktion trotz Störung
	MethodCall_InitStateDrive : BOOL;
	InputVar_InitStateDrive : BOOL;
END_VAR
VAR
	bFirstScan : BOOL := TRUE;
	FirstScanCount: INT := 0;
	AlwaysTrue : BOOL := TRUE;
	TestingVariable : BOOL;	
	 nTaskIdx : DINT;
	RS_InitialState: RS;
	RS_InitialState11: RS;	
	RS_InitialDrive: RS;
	RS_ManualOperationMode: RS;
	RS_AutomaticOperationMode: RS;
	RS_CycleEnded: RS;
	//Count: INT := 0;
	R_TRIG_Manual: R_TRIG;
	R_TRIG_Automatic: R_TRIG;
	R_TRIG_InitialDrive: R_TRIG;
	R_TRIG_CycleEnded: R_TRIG;
	R_TRIG_Init: R_TRIG;
	NeverTrue: BOOL := FALSE;
	SR_D1: SR;
	RS_D2: RS;
	
	RS_D3: RS;
	RS_A5: RS;
	
	
	bFirstCycle: BOOL;
END_VAR
VAR // added by the converter: edge detectors and wires of the graphical bodies
    _w1, _w2, _w3, _w4 : BOOL;
END_VAR

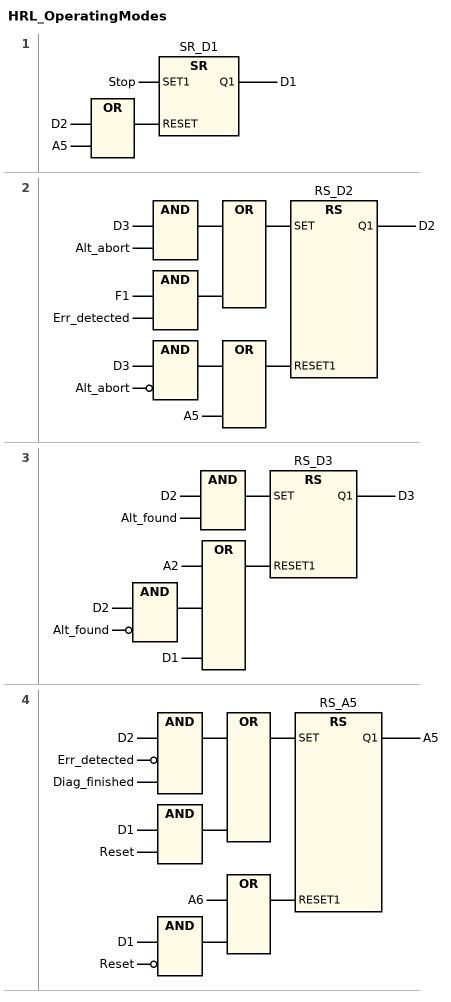
// NETWORK 1
SR_D1(SET1 := Stop, RESET := D2 OR A5); // SR
D1 := SR_D1.Q1;

// NETWORK 2
RS_D2(SET := D3 AND Alt_abort OR F1 AND Err_detected, RESET1 := D3 AND NOT Alt_abort OR A5); // RS
D2 := RS_D2.Q1;

// NETWORK 3
RS_D3(SET := D2 AND Alt_found, RESET1 := A2 OR D2 AND NOT Alt_found OR D1); // RS
D3 := RS_D3.Q1;

// NETWORK 4
RS_A5(SET := D2 AND NOT Err_detected AND Diag_finished OR D1 AND Reset, RESET1 := A6 OR D1 AND NOT Reset); // RS
A5 := RS_A5.Q1;

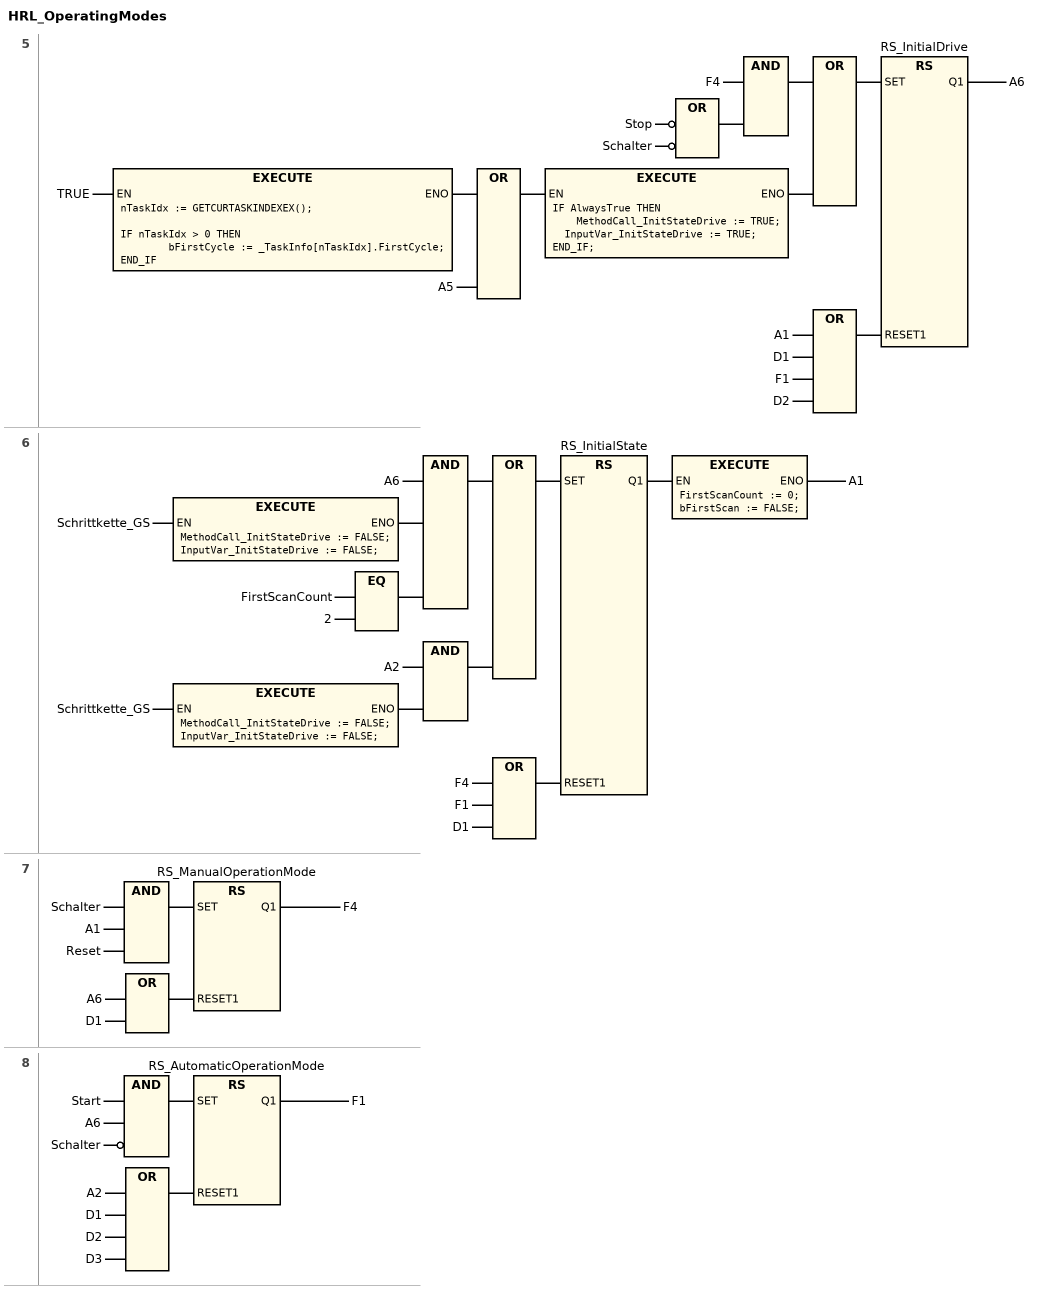
// NETWORK 5
nTaskIdx := GETCURTASKINDEXEX();

IF nTaskIdx > 0 THEN
        bFirstCycle := _TaskInfo[nTaskIdx].FirstCycle;
END_IF
_w1 := TRUE OR A5;
IF _w1 THEN
    IF AlwaysTrue THEN
        MethodCall_InitStateDrive := TRUE;
    	InputVar_InitStateDrive := TRUE;
    END_IF;
END_IF
RS_InitialDrive(SET := F4 AND (NOT Stop OR NOT Schalter) OR _w1, RESET1 := A1 OR D1 OR F1 OR D2); // RS
A6 := RS_InitialDrive.Q1;

// NETWORK 6
_w2 := Schrittkette_GS;
IF _w2 THEN
    MethodCall_InitStateDrive := FALSE;
    InputVar_InitStateDrive := FALSE;
END_IF
_w3 := Schrittkette_GS;
IF _w3 THEN
    MethodCall_InitStateDrive := FALSE;
    InputVar_InitStateDrive := FALSE;
END_IF
RS_InitialState(SET := A6 AND _w2 AND FirstScanCount = 2 OR A2 AND _w3, RESET1 := F4 OR F1 OR D1); // RS
_w4 := RS_InitialState.Q1;
IF _w4 THEN
    FirstScanCount := 0;
    bFirstScan := FALSE;
END_IF
A1 := _w4;

// NETWORK 7
RS_ManualOperationMode(SET := Schalter AND A1 AND Reset, RESET1 := A6 OR D1); // RS
F4 := RS_ManualOperationMode.Q1;

// NETWORK 8
RS_AutomaticOperationMode(SET := Start AND A6 AND NOT Schalter, RESET1 := A2 OR D1 OR D2 OR D3); // RS
F1 := RS_AutomaticOperationMode.Q1;

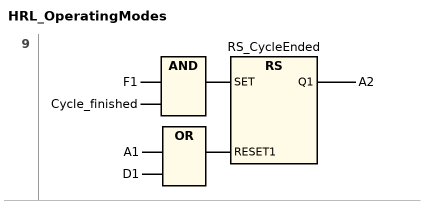
// NETWORK 9
RS_CycleEnded(SET := F1 AND Cycle_finished, RESET1 := A1 OR D1); // RS
A2 := RS_CycleEnded.Q1;

END_FUNCTION_BLOCK

// ---- POUs/DiagnosisHandler/HRL_DiagnosisHandler.TcPOU
FUNCTION_BLOCK HRL_DiagnosisHandler
VAR_INPUT
    Diagnose_gefordert : BOOL;
    ErrorDetectedRaw   : BOOL;
    Reset              : BOOL;
    PulseTime          : TIME := T#100MS;
END_VAR
VAR_OUTPUT
    Err_detected  : BOOL := FALSE;
    Diag_finished : BOOL := FALSE;
    Alt_found     : BOOL := FALSE;
    Busy          : BOOL := FALSE;
END_VAR
VAR
    rtReq      : R_TRIG;
    rtError    : R_TRIG;
    rtDiagAck  : R_TRIG;
    rtAltFound : R_TRIG;
    tpPulse    : TP;
END_VAR

rtReq(CLK := Diagnose_gefordert);
rtError(CLK := ErrorDetectedRaw);
rtDiagAck(CLK := OPCUA.Diag_finished);
rtAltFound(CLK := OPCUA.Alt_found);

IF Reset THEN
    Err_detected := FALSE;
    Diag_finished := FALSE;
    Alt_found := FALSE;
    Busy := FALSE;
    OPCUA.TriggerD2 := FALSE;
END_IF

IF rtError.Q THEN
    Err_detected := TRUE;
    Diag_finished := FALSE;
    Alt_found := FALSE;
END_IF

tpPulse(
    IN := rtReq.Q AND Err_detected AND NOT Busy,
    PT := PulseTime
);

IF rtReq.Q AND Err_detected AND NOT Busy THEN
    Busy := TRUE;
END_IF

IF tpPulse.Q THEN
    OPCUA.TriggerD2 := TRUE;
ELSIF OPCUA.TriggerD2 AND Diag_finished THEN
    OPCUA.TriggerD2 := FALSE;
END_IF

IF Busy AND rtDiagAck.Q THEN
    Diag_finished := TRUE;
    Alt_found := FALSE;
    Busy := FALSE;
    OPCUA.Diag_finished := FALSE;
    OPCUA.TriggerD2 := FALSE;
END_IF

IF Busy AND rtAltFound.Q THEN
    Alt_found := TRUE;
    Diag_finished := TRUE;
    Busy := FALSE;
    OPCUA.Alt_found := FALSE;
    OPCUA.TriggerD2 := FALSE;
END_IF

IF NOT Diagnose_gefordert AND (Diag_finished OR Alt_found) THEN
    Err_detected := FALSE;
    Diag_finished := FALSE;
    Alt_found := FALSE;
END_IF

END_FUNCTION_BLOCK

// ---- POUs/InitStateDrive/HRL_RGB_InitialStateDrive.TcPOU
FUNCTION_BLOCK HRL_RGB_InitialStateDrive
VAR_INPUT
	MethodCall_InitDrive		: BOOL;
	ESS							: BOOL;
	InputInitDriveMode			: BOOL;
	TouchSensor01_SRM			: BOOL;
	TouchSensor02_RGB_vertical	: BOOL;
	TouchSensor03_RGB_horizontal: BOOL;
	TOF_Time_TSR				: TIME;
	InitDriveMode 				: BOOL;
END_VAR

VAR_OUTPUT
	SRM_MotorBackwards: BOOL;
	SRM_MotorForwards: BOOL;
	RGB_VerticalUp: BOOL;
	RGB_VerticalDown: BOOL;
	RGB_HorizontalForwards: BOOL;
	RGB_HorizontalBackwards: BOOL;
	ResetMethodCall_SRM	: BOOL;
	ResetMethodCall_RGB_Vertical	: BOOL;
	ResetMethodCall_RGB_Horizontal	: BOOL;
	Count_SRM_MotorBackw : INT;
	Count_SRM_MotorForw : INT;
END_VAR
VAR
	TSR : BOOL := TRUE;
	DirectionVerticalSRM : BOOL := TRUE;
	DirectionVertical : BOOL := TRUE;
	DirectionHorizontal : BOOL := TRUE;
	
	HRL_RGB_SRM_InitDrive: AxisControl_MultipleInputSensors;
	HRL_RGB_Vertical_InitDrive: AxisControl_MultipleInputSensors;
	HRL_RGB_Horizontal_InitDrive: AxisControl_MultipleInputSensors;
END_VAR

HRL_RGB_SRM_InitDrive(
    MethodCall := MethodCall_InitDrive,
    EmergencyStopSignal := ESS,
    Direction := DirectionVerticalSRM,
    InitStateDrive_Input := InputInitDriveMode,
    DI01 := FALSE,
    DI02 := TouchSensor01_SRM,
    TouchSensorRelief := TSR,
    TOF_Time_MotorControl := T#0MS,
    TOF_Time_TouchSensorRelief := TOF_Time_TSR,
    OperatingMode := InitDriveMode
);
SRM_MotorBackwards := HRL_RGB_SRM_InitDrive.DigitalOutputControl_01;

HRL_RGB_Vertical_InitDrive(
    MethodCall := MethodCall_InitDrive,
    EmergencyStopSignal := ESS,
    Direction := DirectionVertical,
    InitStateDrive_Input := InputInitDriveMode,
    DI01 := FALSE,
    DI02 := TouchSensor02_RGB_vertical,
    TouchSensorRelief := TSR,
    TOF_Time_MotorControl := T#0MS,
    TOF_Time_TouchSensorRelief := TOF_Time_TSR,
    OperatingMode := InitDriveMode
);
RGB_VerticalUp := HRL_RGB_Vertical_InitDrive.DigitalOutputControl_01;

HRL_RGB_Horizontal_InitDrive(
    MethodCall := MethodCall_InitDrive,
    EmergencyStopSignal := ESS,
    Direction := DirectionHorizontal,
    InitStateDrive_Input := InputInitDriveMode,
    DI01 := FALSE,
    DI02 := TouchSensor03_RGB_horizontal,
    TouchSensorRelief := TSR,
    TOF_Time_MotorControl := T#0MS,
    TOF_Time_TouchSensorRelief := TOF_Time_TSR,
    OperatingMode := InitDriveMode
);
RGB_HorizontalBackwards := HRL_RGB_Horizontal_InitDrive.DigitalOutputControl_01;

END_FUNCTION_BLOCK

// ---- POUs/VSG_SkillSet.TcPOU
PROGRAM VSG_SkillSet
VAR
    {attribute 'OPC.UA.DA':= '1'}
    VSG_ErrorDetected : BOOL := FALSE;

    {attribute 'OPC.UA.DA':= '1'}
    VSG_ErrorCode : UDINT := 0;

    {attribute 'OPC.UA.DA':= '1'}
    VSG_Skill_HorizontalMoveForwards : VSG_AS_HorizontalMoveEncoder;

    {attribute 'OPC.UA.DA':= '1'}
    VSG_Skill_HorizontalMoveBackwards : VSG_AS_HorizontalMoveEncoder;

    {attribute 'OPC.UA.DA':= '1'}
    VSG_Skill_VerticalMoveForwards : VSG_AS_VerticalMoveEncoder;

    {attribute 'OPC.UA.DA':= '1'}
    VSG_Skill_VerticalMoveBackwards : VSG_AS_VerticalMoveEncoder;

    {attribute 'OPC.UA.DA':= '1'}
    VSG_Skill_RotationMoveCW : VSG_AS_RotationMoveEncoder;

    {attribute 'OPC.UA.DA':= '1'}
    VSG_Skill_RotationMoveCCW : VSG_AS_RotationMoveEncoder;

    {attribute 'OPC.UA.DA':= '1'}
    VSG_Skill_SuctionProcess : VSG_AS_CompressorControl;

    VSG_ControlOfOutputs : VSG_ControlOfOutputs;
    VSG_OperatingModes : VSG_OperatingModes;
    VSG_DiagnosisHandler : VSG_DiagnosisHandler;
    VSG_InitialStateDrive : VSG_InitialStateDrive;
    bSuctionTrackingLatched : BOOL := FALSE;

    VSG_MoveHorizontalForwards01 : BOOL;
    VSG_MoveHorizontalForwards02 : BOOL;
    VSG_MoveHorizontalBackwards01 : BOOL;
    VSG_MoveHorizontalBackwards02 : BOOL;

    VSG_MoveVerticalDown01 : BOOL;
    VSG_MoveVerticalDown02 : BOOL;
    VSG_MoveVerticalUp01 : BOOL;
    VSG_MoveVerticalUp02 : BOOL;

    VSG_MoveRotationCW01 : BOOL;
    VSG_MoveRotationCW02 : BOOL;
    VSG_MoveRotationCCW01 : BOOL;
    VSG_MoveRotationCCW02 : BOOL;

    VSG_Compressor : BOOL;
    VSG_Valve : BOOL;

    Init_VSG_VertikalUp : BOOL;
    Init_VSG_VertikalDown : BOOL;
    Init_VSG_HorizontalForwards : BOOL;
    Init_VSG_HorizontalBackwards : BOOL;
    Init_VSG_RotationCW : BOOL;
    Init_VSG_RotationCCW : BOOL;

    ResetButton : BOOL;
    StartButton : BOOL;
    ConfirmationButton : BOOL;

    TIME_TSR : TIME := T#150MS;

    MethodCall_InitStateDrive : BOOL;
    InputVar_InitStateDrive : BOOL;
	sCurrentGemmaState: STRING(80);
	sLastNonFailureGemmaState : STRING(80) := '';
    rtD2 : R_TRIG;
END_VAR

IF GVL_Sim.bSimMode THEN

    GVL.diNotAus_Kanal_A := GVL_Sim.diNotAus_Kanal_A;
    GVL.diNotAus_Kanal_B := GVL_Sim.diNotAus_Kanal_B;

    GVL_VSG.VSG_Enc_vertikal_I1 := GVL_VSG_Sim.VSG_Enc_vertikal_I1;
    GVL_VSG.VSG_Enc_vertikal_I2 := GVL_VSG_Sim.VSG_Enc_vertikal_I2;

    GVL_VSG.VSG_Enc_horizontal_I1 := GVL_VSG_Sim.VSG_Enc_horizontal_I1;
    GVL_VSG.VSG_Enc_horizontal_I2 := GVL_VSG_Sim.VSG_Enc_horizontal_I2;

    GVL_VSG.VSG_Enc_drehen_I1 := GVL_VSG_Sim.VSG_Enc_drehen_I1;
    GVL_VSG.VSG_Enc_drehen_I2 := GVL_VSG_Sim.VSG_Enc_drehen_I2;

    GVL_VSG.VSG_Ref_Schalter_vertikal := GVL_VSG_Sim.VSG_Ref_Schalter_vertikal;
    GVL_VSG.VSG_Ref_Schalter_horizontal := GVL_VSG_Sim.VSG_Ref_Schalter_horizontal;
    GVL_VSG.VSG_Ref_Schalter_drehen := GVL_VSG_Sim.VSG_Ref_Schalter_drehen;

END_IF;


VSG_OperatingModes(
    Start := StartButton,
    Stop := NOT ((GVL.diNotAus_Kanal_A) AND (GVL.diNotAus_Kanal_B)),
    Reset := ResetButton,
    Schalter := ConfirmationButton,

    Schrittkette_GS :=
        VSG_InitialStateDrive.ResetMethodCall_RGB_Horizontal
        AND VSG_InitialStateDrive.ResetMethodCall_RGB_Vertical
        AND VSG_InitialStateDrive.ResetMethodCall_RotateCW,

    Count1 := 0,
    Count2 := 0,

    Alt_abort := OPCUA.Alt_abort,
    Err_detected := VSG_DiagnosisHandler.Err_detected,
    Diag_finished := VSG_DiagnosisHandler.Diag_finished,
    Alt_found := VSG_DiagnosisHandler.Alt_found,
    Cycle_finished := OPCUA.Cycle_finished
);


VSG_InitialStateDrive(
    MethodCall_InitDrive := MethodCall_InitStateDrive,
    ESS := ((GVL.diNotAus_Kanal_A) AND (GVL.diNotAus_Kanal_B)),
    InputInitDriveMode := InputVar_InitStateDrive,
    TouchSensor01_Rotation := GVL_VSG.VSG_Ref_Schalter_drehen,
    TouchSensor02_Vertical := GVL_VSG.VSG_Ref_Schalter_vertikal,
    TouchSensor03_horizontal := GVL_VSG.VSG_Ref_Schalter_horizontal,
    TOF_Time_TSR := TIME_TSR,
    InitDriveMode := VSG_OperatingModes.A6
);

Init_VSG_RotationCW := VSG_InitialStateDrive.VSG_Init_RotateCW;
Init_VSG_VertikalUp := VSG_InitialStateDrive.VSG_Init_VerticalUp;
Init_VSG_HorizontalBackwards := VSG_InitialStateDrive.VSG_Init_HorizontalBackwards;


VSG_Skill_HorizontalMoveForwards(
    ESS := ((GVL.diNotAus_Kanal_A) AND (GVL.diNotAus_Kanal_B)),
    TouchSensor01 := GVL_VSG.VSG_Ref_Schalter_horizontal,
    EncoderStartPosition01 := GVL_VSG.VSG_Enc_horizontal_I1,
    EncoderStartPosition02 := GVL_VSG.VSG_Enc_horizontal_I2,
    TOF_Time_TSR := TIME_TSR,
    AutomaticMode := VSG_OperatingModes.A6
);

VSG_MoveHorizontalForwards01 := VSG_Skill_HorizontalMoveForwards.DO_MovingHorizontalVSG_01;


VSG_Skill_HorizontalMoveBackwards(
    ESS := ((GVL.diNotAus_Kanal_A) AND (GVL.diNotAus_Kanal_B)),
    TouchSensor01 := GVL_VSG.VSG_Ref_Schalter_horizontal,
    EncoderStartPosition01 := GVL_VSG.VSG_Enc_horizontal_I1,
    EncoderStartPosition02 := GVL_VSG.VSG_Enc_horizontal_I2,
    TOF_Time_TSR := TIME_TSR,
    AutomaticMode := VSG_OperatingModes.A6
);

VSG_MoveHorizontalBackwards02 := VSG_Skill_HorizontalMoveBackwards.DO_MovingHorizontalVSG_01;


VSG_Skill_VerticalMoveForwards(
    ESS := ((GVL.diNotAus_Kanal_A) AND (GVL.diNotAus_Kanal_B)),
    TouchSensor01 := GVL_VSG.VSG_Ref_Schalter_vertikal,
    EncoderStartPosition01 := GVL_VSG.VSG_Enc_vertikal_I1,
    EncoderStartPosition02 := GVL_VSG.VSG_Enc_vertikal_I2,
    TOF_Time_TSR := TIME_TSR,
    AutomaticMode := VSG_OperatingModes.A6
);

VSG_MoveVerticalDown01 := VSG_Skill_VerticalMoveForwards.DO_MovingVerticalVSG_01;


VSG_Skill_VerticalMoveBackwards(
    ESS := ((GVL.diNotAus_Kanal_A) AND (GVL.diNotAus_Kanal_B)),
    TouchSensor01 := GVL_VSG.VSG_Ref_Schalter_vertikal,
    EncoderStartPosition01 := GVL_VSG.VSG_Enc_vertikal_I1,
    EncoderStartPosition02 := GVL_VSG.VSG_Enc_vertikal_I2,
    TOF_Time_TSR := TIME_TSR,
    AutomaticMode := VSG_OperatingModes.A6
);

VSG_MoveVerticalUp02 := VSG_Skill_VerticalMoveBackwards.DO_MovingVerticalVSG_01;


VSG_Skill_RotationMoveCW(
    ESS := ((GVL.diNotAus_Kanal_A) AND (GVL.diNotAus_Kanal_B)),
    TouchSensor01 := GVL_VSG.VSG_Ref_Schalter_drehen,
    EncoderStartPosition01 := GVL_VSG.VSG_Enc_drehen_I1,
    EncoderStartPosition02 := GVL_VSG.VSG_Enc_drehen_I2,
    TOF_Time_TSR := TIME_TSR,
    AutomaticMode := VSG_OperatingModes.A6
);

VSG_MoveRotationCW01 := VSG_Skill_RotationMoveCW.DO_MovingRotationVSG_01;


VSG_Skill_RotationMoveCCW(
    ESS := ((GVL.diNotAus_Kanal_A) AND (GVL.diNotAus_Kanal_B)),
    TouchSensor01 := GVL_VSG.VSG_Ref_Schalter_drehen,
    EncoderStartPosition01 := GVL_VSG.VSG_Enc_drehen_I1,
    EncoderStartPosition02 := GVL_VSG.VSG_Enc_drehen_I2,
    TOF_Time_TSR := TIME_TSR,
    AutomaticMode := VSG_OperatingModes.A6
);

VSG_MoveRotationCCW02 := VSG_Skill_RotationMoveCCW.DO_MovingRotationVSG_01;


VSG_Skill_SuctionProcess(
    ESS := ((GVL.diNotAus_Kanal_A) AND (GVL.diNotAus_Kanal_B)),

    EncoderStartPosition01 := GVL_VSG.VSG_Enc_drehen_I1,
    EncoderStartPosition02 := GVL_VSG.VSG_Enc_drehen_I2,
    EncoderStartPosition03 := GVL_VSG.VSG_Enc_horizontal_I1,
    EncoderStartPosition04 := GVL_VSG.VSG_Enc_horizontal_I2,
    EncoderStartPosition05 := GVL_VSG.VSG_Enc_vertikal_I1,
    EncoderStartPosition06 := GVL_VSG.VSG_Enc_vertikal_I2,

    WorkpieceAtPickupPosition := GVL_HRL.HRL_LS_aussen,

    AutomaticMode := VSG_OperatingModes.F1 AND NOT VSG_OperatingModes.D2
);

VSG_Compressor := VSG_Skill_SuctionProcess.DO_CompressorVSG;
VSG_Valve := VSG_Skill_SuctionProcess.DO_ValveVSG;

VSG_ErrorDetected := VSG_Skill_SuctionProcess.VSG_ErrorDetected;
VSG_ErrorCode := VSG_Skill_SuctionProcess.VSG_ErrorCode;


VSG_DiagnosisHandler(
    Diagnose_gefordert := VSG_OperatingModes.D2,
    ErrorDetectedRaw := VSG_Skill_SuctionProcess.VSG_ErrorDetected,
    Reset := ResetButton
);


VSG_ControlOfOutputs(
    F4 := VSG_OperatingModes.F4,
    F1 := VSG_OperatingModes.F1,
    A2 := VSG_OperatingModes.A2,
    A1 := VSG_OperatingModes.A1,
    A6 := VSG_OperatingModes.A6,
    Start := VSG_OperatingModes.Start,

    VSG_VertikalDown01 := VSG_MoveVerticalDown01,
    VSG_VertikalDown02 := VSG_MoveVerticalDown02,
    VSG_VertikalUp01 := VSG_MoveVerticalUp01,
    VSG_VertikalUp02 := VSG_MoveVerticalUp02,

    VSG_HorizontalForwards01 := VSG_MoveHorizontalForwards01,
    VSG_HorizontalForwards02 := VSG_MoveHorizontalForwards02,
    VSG_HorizontalBackwards01 := VSG_MoveHorizontalBackwards01,
    VSG_HorizontalBackwards02 := VSG_MoveHorizontalBackwards02,

    VSG_RotationCW01 := VSG_MoveRotationCW01,
    VSG_RotationCW02 := VSG_MoveRotationCW02,
    VSG_RotationCCW01 := VSG_MoveRotationCCW01,
    VSG_RotationCCW02 := VSG_MoveRotationCCW02,

    VSG_Compressor := VSG_Compressor,
    VSG_Valve := VSG_Valve,

    Init_VSG_VertikalUp := Init_VSG_VertikalUp,
    Init_VSG_VertikalDown := Init_VSG_VertikalDown,
    Init_VSG_HorizontalForwards := Init_VSG_HorizontalForwards,
    Init_VSG_HorizontalBackwards := Init_VSG_HorizontalBackwards,
    Init_VSG_RotationCW := Init_VSG_RotationCW,
    Init_VSG_RotationCCW := Init_VSG_RotationCCW
);


IF GVL_Sim.bSimMode THEN

    GVL_VSG_Sim.VSG_MOT_vertikal_runter := VSG_ControlOfOutputs.MoveVerticalDown;
    GVL_VSG_Sim.VSG_MOT_vertikal_hoch := VSG_ControlOfOutputs.MoveVerticalUp;

    GVL_VSG_Sim.VSG_MOT_horizontal_vorwaerts := VSG_ControlOfOutputs.MoveHorizontalForwards;
    GVL_VSG_Sim.VSG_MOT_horizontal_rueckwaerts := VSG_ControlOfOutputs.MoveHorizontalBackwards;

    GVL_VSG_Sim.VSG_MOT_drehen_CW := VSG_ControlOfOutputs.MoveRotationCW;
    GVL_VSG_Sim.VSG_MOT_drehen_CCW := VSG_ControlOfOutputs.MoveRotationCCW;

    GVL_VSG_Sim.VSG_Kompressor := VSG_ControlOfOutputs.CompressorON;
    GVL_VSG_Sim.VSG_MV_Vakuum := VSG_ControlOfOutputs.ValveON;

ELSE

    GVL_VSG.VSG_MOT_vertikal_runter := VSG_ControlOfOutputs.MoveVerticalDown;
    GVL_VSG.VSG_MOT_vertikal_hoch := VSG_ControlOfOutputs.MoveVerticalUp;

    GVL_VSG.VSG_MOT_horizontal_vorwaerts := VSG_ControlOfOutputs.MoveHorizontalForwards;
    GVL_VSG.VSG_MOT_horizontal_rueckwaerts := VSG_ControlOfOutputs.MoveHorizontalBackwards;

    GVL_VSG.VSG_MOT_drehen_CW := VSG_ControlOfOutputs.MoveRotationCW;
    GVL_VSG.VSG_MOT_drehen_CCW := VSG_ControlOfOutputs.MoveRotationCCW;

    GVL_VSG.VSG_Kompressor := VSG_ControlOfOutputs.CompressorON;
    GVL_VSG.VSG_MV_Vakuum := VSG_ControlOfOutputs.ValveON;

END_IF;

//GEMMA_Mappings
IF VSG_OperatingModes.A1 THEN
    sCurrentGemmaState := 'VSG_OperatingModes.A1';
ELSIF VSG_OperatingModes.A2 THEN
    sCurrentGemmaState := 'VSG_OperatingModes.A2';
ELSIF VSG_OperatingModes.A5 THEN
    sCurrentGemmaState := 'VSG_OperatingModes.A5';
ELSIF VSG_OperatingModes.A6 THEN
    sCurrentGemmaState := 'VSG_OperatingModes.A6';
ELSIF VSG_OperatingModes.F1 THEN
    sCurrentGemmaState := 'VSG_OperatingModes.F1';
ELSIF VSG_OperatingModes.F4 THEN
    sCurrentGemmaState := 'VSG_OperatingModes.F4';
ELSIF VSG_OperatingModes.D1 THEN
    sCurrentGemmaState := 'VSG_OperatingModes.D1';
ELSIF VSG_OperatingModes.D3 THEN
    sCurrentGemmaState := 'VSG_OperatingModes.D3';
END_IF;

IF NOT VSG_OperatingModes.D2 THEN
    sLastNonFailureGemmaState := sCurrentGemmaState;
END_IF;

rtD2(CLK := VSG_OperatingModes.D2);

IF rtD2.Q THEN
    OPCUA.LastGEMMAStateBeforeFailure := sLastNonFailureGemmaState;
END_IF;

END_PROGRAM

// ---- POUs/Moduls/VSG_Skills/VSG_AS_HorizontalMoveEncoder.TcPOU
{attribute 'OPC.UA.DA.JobMethod' := 'JobMethode_HorizontalMove'}
FUNCTION_BLOCK VSG_AS_HorizontalMoveEncoder
VAR
    MethodCall_HorizontalMove : BOOL := FALSE;
    ResetMethodCall : BOOL := FALSE;

    DirectionHorizontal : BOOL := TRUE;

    EncoderTargetPosition01 : UDINT;
    EncoderTargetPosition02 : UDINT;

    TSR : BOOL := FALSE;

    callCounterStart : ULINT;
    callCounterCheckState : ULINT;
    callCounterAbort : ULINT;

    jobRunning : BOOL := FALSE;
    jobFinished : BOOL := FALSE;
    state : UDINT := 0;

    VSG_HorizontalMoveWithEncoder : AxisControl_Encoder;
END_VAR

VAR_INPUT
    ESS : BOOL;
    TouchSensor01 : BOOL;
    EncoderStartPosition01 : UDINT;
    EncoderStartPosition02 : UDINT;
    TOF_Time_TSR : TIME;
    AutomaticMode : BOOL;
END_VAR

VAR_OUTPUT
    DO_MovingHorizontalVSG_01 : BOOL;
END_VAR

VSG_HorizontalMoveWithEncoder(
    MethodCall := MethodCall_HorizontalMove,
    EmergencyStopSignal := NOT ESS,
    Direction := DirectionHorizontal,
    InitStateDrive_Input := FALSE,
    DI01 := TouchSensor01,
    DI02_EncoderStart01 := EncoderStartPosition01,
    DI03_EncoderTarget01 := EncoderTargetPosition01,
    DI04_EncoderStart02 := EncoderStartPosition02,
    DI05_EncoderTarget02 := EncoderTargetPosition02,
    TouchSensorRelief := TSR,
    TOF_Time_MotorControl := T#0MS,
    TOF_Time_TouchSensorRelief := TOF_Time_TSR,
    OperatingMode := AutomaticMode
);

DO_MovingHorizontalVSG_01 := VSG_HorizontalMoveWithEncoder.DigitalOutputControl_01;
ResetMethodCall := VSG_HorizontalMoveWithEncoder.ResetMethodCall;

IF ResetMethodCall THEN
    MethodCall_HorizontalMove := FALSE;
    jobRunning := FALSE;
    jobFinished := TRUE;
    state := 100;
END_IF;

{attribute 'TcRpcEnable' := '1'}
METHOD Abort : HRESULT
VAR_INPUT
    hdl : UDINT;
END_VAR
callCounterAbort := callCounterAbort + 1;

MethodCall_HorizontalMove := FALSE;
DO_MovingHorizontalVSG_01 := FALSE;

jobRunning := FALSE;
jobFinished := TRUE;
state := 999;

Abort := 0;
END_METHOD

{attribute 'TcRpcEnable' := '1'}
METHOD CheckState : HRESULT
VAR_INPUT
    hdl : UDINT;
END_VAR

VAR_OUTPUT
    bBusy : BOOL;
    State : UDINT;
    IsDone : BOOL;
END_VAR
callCounterCheckState := callCounterCheckState + 1;

bBusy := jobRunning;
State := state;
IsDone := jobFinished;

CheckState := 0;
END_METHOD

{attribute 'TcRpcEnable' := '1'}
METHOD Start : HRESULT
VAR_INPUT
    MethodCall : BOOL;
    MovementDirection : BOOL;
    EncoderPositionHorizontal_01 : UDINT;
    EncoderPositionHorizontal_02 : UDINT;
    TouchSensorRelief : BOOL;
END_VAR

VAR_OUTPUT
    hdl : UDINT;
END_VAR
callCounterStart := callCounterStart + 1;

IF NOT jobRunning THEN

    MethodCall_HorizontalMove := MethodCall;
    DirectionHorizontal := MovementDirection;

    EncoderTargetPosition01 := EncoderPositionHorizontal_01;
    EncoderTargetPosition02 := EncoderPositionHorizontal_02;

    TSR := TouchSensorRelief;

    jobRunning := TRUE;
    jobFinished := FALSE;
    state := 1;

    hdl := 1;
    Start := 0;

ELSE

    hdl := 0;
    Start := 16#800700AA;

END_IF;
END_METHOD

END_FUNCTION_BLOCK

// ---- POUs/Moduls/VSG_Skills/VSG_AS_VerticalMoveEncoder.TcPOU
{attribute 'OPC.UA.DA.JobMethod' := 'JobMethode_VerticalMove'}
FUNCTION_BLOCK VSG_AS_VerticalMoveEncoder
VAR
    MethodCall_VerticalMove : BOOL := FALSE;
    ResetMethodCall : BOOL := FALSE;

    DirectionVertical : BOOL := TRUE;

    EncoderTargetPosition01 : UDINT;
    EncoderTargetPosition02 : UDINT;

    TSR : BOOL := FALSE;

    callCounterStart : ULINT;
    callCounterCheckState : ULINT;
    callCounterAbort : ULINT;

    jobRunning : BOOL := FALSE;
    jobFinished : BOOL := FALSE;
    state : UDINT := 0;

    VSG_VerticalMoveWithEncoder : AxisControl_Encoder;
END_VAR

